// TwinCAT 3 PLC project mobject_graph
// Title: mobject-graph
// Company: mobject
// Author: mobject dev team
// ProjectVersion: 0.12.0
// ProgramVersion: 3.1.4024.0
// libraries:
//   Tc2_Standard, * (Beckhoff Automation GmbH)
//   Tc2_System, * (Beckhoff Automation GmbH)
//   Tc2_Utilities, * (Beckhoff Automation GmbH)
//   mobject-core,0.4.0,mobject
//   mobject-server,0.14.0,mobject
// project tree:
//   Alarms/Base/ Alarm.TcPOU
//   Alarms/ DeserializationFailedAlarm.TcPOU, DeserializationFailedNodeNotSupportedAlarm.TcPOU, FunctionFailedAlarm.TcPOU
//   Alarms/Events/ AlarmAddedEvent.TcPOU (not stored), I_AlarmAddedEvent.TcIO
//   Alarms/Host/ AlarmHost.TcPOU
//   Alarms/Interfaces/ I_Alarm.TcIO (not stored), I_Alarms.TcIO, I_HostAlarms.TcIO
//   API/ GraphFrameworkApi.TcPOU
//   API/Handlers/ CreateGraphMultiUserRpcHandler.TcPOU, CreateGraphRpcHandler.TcPOU, GetBlueprintsRpcHandler.TcPOU, GetContentValueHandler.TcPOU, UpdateParameterValueHandler.TcPOU, GetStatusRpcHandler.TcPOU
//   API/Visitors/ GetBlueprintsVisitor.TcPOU, GetStatusVisitor.TcPOU, IncludeInGetStatusVisitor.TcPOU, RetrieveNodeContentValue.TcPOU
//   Content/Base/ Content.TcPOU
//   Content/Events/ ContentAddedEvent.TcPOU (not stored), I_ContentAddedEvent.TcIO
//   Content/Host/ ContentHost.TcPOU
//   Content/Interface/ I_Content.TcIO (not stored), I_Contents.TcIO, I_HostContent.TcIO (not stored)
//   Errors/ MissingNodePrototypeDeserializationError.TcPOU (not stored)
//   Extensions/Base/ Extension.TcPOU
//   Extensions/Events/ ExtensionAddedEvent.TcPOU, I_ExtensionAddedEvent.TcIO (not stored)
//   Extensions/Host/ ExtensionHost.TcPOU
//   Extensions/Interface/ I_Extension.TcIO, I_Extensions.TcIO, I_HostExtensions.TcIO (not stored)
//   Extensions/Namespace/ ExtensionNamespace.TcPOU (not stored)
//   Extensions/PreExecutionCheck/Alarms/ PreExecutionCheckFailedAlarm.TcPOU
//   Extensions/PreExecutionCheck/Checks/ I_PreExecutionChecks.TcIO, PreExecutionChecks.TcPOU
//   Extensions/PreExecutionCheck/Interfaces/ I_PreCheckedNode.TcIO (not stored)
//   Extensions/PreExecutionCheck/ PreExecutionCheckExtension.TcPOU
//   GraphFramework/ GraphFramework.TcPOU
//   GraphFramework/Interface/ I_GraphFramework.TcIO
//   Graph/Base/ Graph.TcPOU
//   Graph/Events/ GraphAddedEvent.TcPOU (not stored), I_GraphAddedEvent.TcIO
//   Graph/Host/ GraphHost.TcPOU
//   Graph/Interfaces/ I_Graph.TcIO (not stored), I_Graphs.TcIO (not stored), I_HostGraphs.TcIO (not stored)
//   IecDatatypesPack/ IecDatatypesPack.TcPOU
//   InputPort/Base/ InputPort.TcPOU
//   InputPort/Events/ InputPortAddedEvent.TcPOU (not stored), InputPortChangedEvent.TcPOU (not stored), I_InputPortAddedEvent.TcIO (not stored), I_InputPortChangedEvent.TcIO (not stored)
//   InputPort/Host/ InputPortHost.TcPOU
//   InputPort/Interface/ I_HostInputPorts.TcIO, I_InputPort.TcIO (not stored), I_InputPorts.TcIO
//   Metadata/Base/ Metadata.TcPOU
//   Metadata/Events/ I_MetadataAddedEvent.TcIO, MetadataAddedEvent.TcPOU (not stored)
//   Metadata/Host/ MetadataHost.TcPOU
//   Metadata/Interface/ I_HostMetadata.TcIO, I_Metadata.TcIO, I_Metadatum.TcIO
//   NodeFactory/Base/ NodeFactory.TcPOU
//   NodeFactory/Datatype/ DatatypeNodeFactory.TcPOU
//   NodeFactory/Interface/ I_NodeFactory.TcIO (not stored)
//   NodePrototype/Base/ NodePrototype.TcPOU (not stored)
//   NodePrototype/Host/ NodePrototypeHost.TcPOU
//   NodePrototype/Interface/ I_NodePrototype.TcIO (not stored), I_NodePrototypes.TcIO
//   Node/Base/ Node.TcPOU
//   Node/Bundle/ AnyAliasArrayBundleNode.TcPOU, AnyStructureBundleNode.TcPOU, AnyArrayBundleNode.TcPOU, AnyAliasStructureBundleNode.TcPOU
//   Node/Events/ I_NodeAddedEvent.TcIO, I_NodeExecuteBeginEvent.TcIO, I_NodeExecuteEndEvent.TcIO, I_NodePreExecuteEvent.TcIO, NodeAddedEvent.TcPOU, NodeExecuteBeginEvent.TcPOU, NodeExecuteEndEvent.TcPOU, NodePreExecuteEvent.TcPOU
//   Node/Unbundle/ AnyAliasArrayUnbundleNode.TcPOU, AnyStructureUnbundleNode.TcPOU (not stored), AnyArrayUnbundleNode.TcPOU, AnyAliasStructureUnbundleNode.TcPOU
//   Node/Display/ AnyDisplayNode.TcPOU (not stored)
//   Node/Host/ NodeHost.TcPOU
//   Node/Interface/ I_HostNodes.TcIO (not stored), I_Node.TcIO, I_Nodes.TcIO
//   Node/Literal/ AnyLiteralNode.TcPOU (not stored)
//   OutputPort/Base/ OutputPort.TcPOU
//   OutputPort/Events/ I_OutputPortAddedEvent.TcIO, I_OutputPortChangedEvent.TcIO (not stored), OutputPortAddedEvent.TcPOU (not stored), OutputPortChangedEvent.TcPOU (not stored)
//   OutputPort/Host/ OutputPortHost.TcPOU
//   OutputPort/Interface/ I_HostOutputPorts.TcIO, I_OutputPort.TcIO (not stored), I_OutputPorts.TcIO
//   Packs/DatatypePack/ I_DatatypePack.TcIO (not stored)
//   Packs/GraphPack/ I_GraphPack.TcIO (not stored)
//   Packs/NodePack/ I_NodePack.TcIO
//   Parameters/Base/ Parameter.TcPOU
//   Parameters/Events/ I_ParameterAddedEvent.TcIO, ParameterAddedEvent.TcPOU
//   Parameters/Host/ ParameterHost.TcPOU
//   Parameters/Interface/ I_HostParameters.TcIO, I_Parameter.TcIO (not stored), I_Parameters.TcIO
//   Visitors/Interfaces/ I_AlarmVisitor.TcIO, I_ContentVisitor.TcIO, I_ExtensionVisitor.TcIO, I_GraphVisitor.TcIO, I_InputPortVisitor.TcIO (not stored), I_MetadataVisitor.TcIO (not stored), I_NodeFactoryVisitor.TcIO, I_NodePrototypeVisitor.TcIO (not stored), I_NodeVisitor.TcIO (not stored), I_OutputPortVisitor.TcIO (not stored), I_ParameterVisitor.TcIO

// ---- Alarms/Events/I_AlarmAddedEvent.TcIO
INTERFACE I_AlarmAddedEvent EXTENDS I_Event

PROPERTY PUBLIC Target : I_Alarm
GET
END_GET
END_PROPERTY

END_INTERFACE

// ---- Alarms/Interfaces/I_Alarms.TcIO
INTERFACE I_Alarms

METHOD PUBLIC Accept
VAR_INPUT
	Visitor : I_AlarmVisitor;
END_VAR
END_METHOD

METHOD AddAlarm
VAR_INPUT
	Alarm : I_Alarm;
END_VAR
END_METHOD

PROPERTY PUBLIC HasAlarms : BOOL
GET
END_GET
END_PROPERTY

PROPERTY PUBLIC HasRaisedAlarm : BOOL
GET
END_GET
END_PROPERTY

END_INTERFACE

// ---- Alarms/Interfaces/I_HostAlarms.TcIO
INTERFACE I_HostAlarms EXTENDS __SYSTEM.IQueryInterface

PROPERTY Alarms : I_Alarms
GET
END_GET
END_PROPERTY

END_INTERFACE

// ---- Content/Events/I_ContentAddedEvent.TcIO
INTERFACE I_ContentAddedEvent EXTENDS I_Event

PROPERTY PUBLIC Target : I_Content
GET
END_GET
END_PROPERTY

END_INTERFACE

// ---- Content/Interface/I_Contents.TcIO
INTERFACE I_Contents

METHOD PUBLIC Accept
VAR_INPUT
	visitor : I_ContentVisitor;
END_VAR
END_METHOD

METHOD AddContent
VAR_INPUT
	Content : I_Content;
END_VAR
END_METHOD

METHOD PUBLIC AddDataAsContent : I_Content
VAR_INPUT
	Name : T_MAXSTRING;
	Data : I_Datatype;
END_VAR
END_METHOD

PROPERTY PUBLIC HasContents : BOOL
GET
END_GET
END_PROPERTY

METHOD PUBLIC TryGetContentByName : BOOL
VAR_INPUT
	Name : T_MAXSTRING;
	Destination : REFERENCE TO I_Content;
END_VAR
END_METHOD

END_INTERFACE

// ---- Extensions/Interface/I_Extension.TcIO
INTERFACE I_Extension EXTENDS I_Disposable, I_HostContent, I_HostInputPorts, I_HostOutputPorts, I_HostAlarms, I_HostParameters, I_HostMetadata, I_EventEmitter, I_Deserializable, I_Serializable

METHOD PUBLIC Accept
VAR_INPUT
	Visitor : I_ExtensionVisitor;
END_VAR
END_METHOD

PROPERTY PUBLIC Name : T_MAXSTRING
GET
END_GET
END_PROPERTY

END_INTERFACE

// ---- Extensions/Interface/I_Extensions.TcIO
INTERFACE I_Extensions

METHOD PUBLIC Accept
VAR_INPUT
	Visitor : I_ExtensionVisitor;
END_VAR
END_METHOD

METHOD AddExtension
VAR_INPUT
	Extension : I_Extension;
END_VAR
END_METHOD

PROPERTY PUBLIC HasExtensions : BOOL
GET
END_GET
END_PROPERTY

METHOD PUBLIC TryGetExtensionByName : BOOL
VAR_INPUT
	Name : T_MAXSTRING;
	Destination : REFERENCE TO I_Extension;
END_VAR
END_METHOD

END_INTERFACE

// ---- Extensions/PreExecutionCheck/Checks/I_PreExecutionChecks.TcIO
INTERFACE I_PreExecutionChecks

METHOD PUBLIC Fail
VAR_INPUT
	Message : T_MAXSTRING;
END_VAR
END_METHOD

PROPERTY PUBLIC Failed : BOOL
GET
END_GET
END_PROPERTY

METHOD PUBLIC IsFalse
VAR_INPUT
	Actual : BOOL;
	Message : T_MAXSTRING;
END_VAR
END_METHOD

METHOD PUBLIC IsTrue
VAR_INPUT
	Actual : BOOL;
	Message : T_MAXSTRING;
END_VAR
END_METHOD

END_INTERFACE

// ---- GraphFramework/Interface/I_GraphFramework.TcIO
INTERFACE I_GraphFramework

METHOD PUBLIC Create : I_Graph
VAR_INPUT
END_VAR
END_METHOD

PROPERTY PUBLIC Datatypes : I_Datatypes
GET
END_GET
END_PROPERTY

PROPERTY PUBLIC NodeFactory : I_NodeFactory
GET
END_GET
END_PROPERTY

END_INTERFACE

// ---- Graph/Events/I_GraphAddedEvent.TcIO
INTERFACE I_GraphAddedEvent EXTENDS I_Event

PROPERTY PUBLIC Target : I_Graph
GET
END_GET
END_PROPERTY

END_INTERFACE

// ---- InputPort/Interface/I_HostInputPorts.TcIO
INTERFACE I_HostInputPorts EXTENDS __SYSTEM.IQueryInterface

PROPERTY InputPorts : I_InputPorts
GET
END_GET
END_PROPERTY

END_INTERFACE

// ---- InputPort/Interface/I_InputPorts.TcIO
INTERFACE I_InputPorts

METHOD PUBLIC Accept
VAR_INPUT
	Visitor : I_InputPortVisitor;
END_VAR
END_METHOD

METHOD PUBLIC AddDataAsInputPort : I_InputPort
VAR_INPUT
	Name : T_MAXSTRING;
	Data : I_Datatype;
END_VAR
END_METHOD

METHOD AddInputPort
VAR_INPUT
	InputPort : I_InputPort;
END_VAR
END_METHOD

PROPERTY PUBLIC HasInputPorts : BOOL
GET
END_GET
END_PROPERTY

METHOD PUBLIC TryGetInputPortByName : BOOL
VAR_INPUT
	Name : T_MAXSTRING;
	Destination : REFERENCE TO I_InputPort;
END_VAR
END_METHOD

END_INTERFACE

// ---- Metadata/Events/I_MetadataAddedEvent.TcIO
INTERFACE I_MetadataAddedEvent EXTENDS I_Event

PROPERTY PUBLIC Target : I_Metadata
GET
END_GET
END_PROPERTY

END_INTERFACE

// ---- Metadata/Interface/I_HostMetadata.TcIO
INTERFACE I_HostMetadata EXTENDS __SYSTEM.IQueryInterface

METHOD PUBLIC AddMetadata : I_HostMetadata
VAR_INPUT
	Name : T_MAXSTRING;
	Data : I_Datatype;
END_VAR
END_METHOD

PROPERTY Metadatum : I_Metadatum
GET
END_GET
END_PROPERTY

END_INTERFACE

// ---- Metadata/Interface/I_Metadata.TcIO
INTERFACE I_Metadata EXTENDS I_Disposable, I_Serializable

METHOD PUBLIC Accept
VAR_INPUT
	Visitor : I_MetadataVisitor;
END_VAR
END_METHOD

PROPERTY PUBLIC Data : I_DataType
GET
END_GET
END_PROPERTY

PROPERTY PUBLIC Name : T_MAXSTRING
GET
END_GET
END_PROPERTY

METHOD PUBLIC SerializeWith
VAR_INPUT
	Serializer : I_Serializer;
END_VAR
END_METHOD

END_INTERFACE

// ---- Metadata/Interface/I_Metadatum.TcIO
INTERFACE I_Metadatum

METHOD PUBLIC Accept
VAR_INPUT
	Visitor : I_MetadataVisitor;
END_VAR
END_METHOD

METHOD PUBLIC AddDataAsMetadata : I_Metadata
VAR_INPUT
	Name : T_MAXSTRING;
	Data : I_Datatype;
END_VAR
END_METHOD

METHOD AddMetadata
VAR_INPUT
	Metadata : I_Metadata;
END_VAR
END_METHOD

PROPERTY PUBLIC HasMetadata : BOOL
GET
END_GET
END_PROPERTY

METHOD PUBLIC TryGetMetadataByName : BOOL
VAR_INPUT
	Name : T_MAXSTRING;
	Destination : REFERENCE TO I_Metadata;
END_VAR
END_METHOD

END_INTERFACE

// ---- NodePrototype/Interface/I_NodePrototypes.TcIO
INTERFACE I_NodePrototypes

METHOD PUBLIC Accept
VAR_INPUT
	Visitor : I_NodePrototypeVisitor;
END_VAR
END_METHOD

PROPERTY PUBLIC HasNodePrototypes : BOOL
GET
END_GET
END_PROPERTY

END_INTERFACE

// ---- Node/Events/I_NodeAddedEvent.TcIO
INTERFACE I_NodeAddedEvent EXTENDS I_Event

PROPERTY PUBLIC Target : I_Node
GET
END_GET
END_PROPERTY

END_INTERFACE

// ---- Node/Events/I_NodeExecuteBeginEvent.TcIO
INTERFACE I_NodeExecuteBeginEvent EXTENDS I_Event

PROPERTY PUBLIC CpuCounterHighBytes : UDINT
GET
END_GET
END_PROPERTY

PROPERTY PUBLIC CpuCounterLowBytes : UDINT
GET
END_GET
END_PROPERTY

PROPERTY PUBLIC Target : I_Node
GET
END_GET
END_PROPERTY

END_INTERFACE

// ---- Node/Events/I_NodeExecuteEndEvent.TcIO
INTERFACE I_NodeExecuteEndEvent EXTENDS I_Event

PROPERTY PUBLIC Target : I_Node
GET
END_GET
END_PROPERTY

END_INTERFACE

// ---- Node/Events/I_NodePreExecuteEvent.TcIO
INTERFACE I_NodePreExecuteEvent EXTENDS I_Event

METHOD PUBLIC Cancel
VAR_INPUT
END_VAR
END_METHOD

PROPERTY PUBLIC ExecuteCancelled : BOOL
GET
END_GET
END_PROPERTY

PROPERTY PUBLIC Target : I_Node
GET
END_GET
END_PROPERTY

END_INTERFACE

// ---- Node/Interface/I_Node.TcIO
INTERFACE I_Node EXTENDS I_Disposable, I_HostContent, I_HostInputPorts, I_HostOutputPorts, I_HostAlarms, I_HostParameters, I_HostExtensions, I_HostMetadata, I_EventEmitter, I_Deserializable, I_Serializable

METHOD PUBLIC Accept
VAR_INPUT
	Visitor : I_NodeVisitor;
END_VAR
END_METHOD

METHOD Clone : I_Node
VAR_INPUT
END_VAR
END_METHOD

METHOD PUBLIC Execute
END_METHOD

PROPERTY PUBLIC Id : T_MAXSTRING
GET
END_GET
END_PROPERTY

PROPERTY PUBLIC Mode : DINT
GET
END_GET
END_PROPERTY

PROPERTY PUBLIC Order : DINT
GET
END_GET
END_PROPERTY

END_INTERFACE

// ---- Node/Interface/I_Nodes.TcIO
INTERFACE I_Nodes

METHOD PUBLIC Accept
VAR_INPUT
	Visitor : I_NodeVisitor;
END_VAR
END_METHOD

METHOD AddNode
VAR_INPUT
	Node : I_Node;
END_VAR
END_METHOD

PROPERTY PUBLIC HasNodes : BOOL
GET
END_GET
END_PROPERTY

METHOD PUBLIC TryGetNodeById : BOOL
VAR_INPUT
	Id : T_MAXSTRING;
	Destination : REFERENCE TO I_Node;
END_VAR
END_METHOD

END_INTERFACE

// ---- OutputPort/Events/I_OutputPortAddedEvent.TcIO
INTERFACE I_OutputPortAddedEvent extends I_Event

PROPERTY PUBLIC Target : I_OutputPort
GET
END_GET
END_PROPERTY

END_INTERFACE

// ---- OutputPort/Interface/I_HostOutputPorts.TcIO
INTERFACE I_HostOutputPorts EXTENDS __SYSTEM.IQueryInterface

PROPERTY OutputPorts : I_OutputPorts
GET
END_GET
END_PROPERTY

END_INTERFACE

// ---- OutputPort/Interface/I_OutputPorts.TcIO
INTERFACE I_OutputPorts

METHOD PUBLIC Accept
VAR_INPUT
	Visitor : I_OutputPortVisitor;
END_VAR
END_METHOD

METHOD PUBLIC AddDataAsOutputPort : I_OutputPort
VAR_INPUT
	Name : T_MAXSTRING;
	Data : I_Datatype;
END_VAR
END_METHOD

METHOD AddOutputPort
VAR_INPUT
	OutputPort : I_OutputPort;
END_VAR
END_METHOD

PROPERTY PUBLIC HasOutputPorts : BOOL
GET
END_GET
END_PROPERTY

METHOD PUBLIC TryGetOutputPortByName : BOOL
VAR_INPUT
	Name : T_MAXSTRING;
	Destination : REFERENCE TO I_OutputPort;
END_VAR
END_METHOD

END_INTERFACE

// ---- Packs/NodePack/I_NodePack.TcIO
INTERFACE I_NodePack

METHOD PUBLIC RegisterWithNodeFactory
VAR_INPUT
	NodeFactory : I_NodeFactory;
END_VAR
END_METHOD

END_INTERFACE

// ---- Parameters/Events/I_ParameterAddedEvent.TcIO
INTERFACE I_ParameterAddedEvent EXTENDS I_Event

PROPERTY PUBLIC TargetParameter : I_Parameter
GET
END_GET
END_PROPERTY

END_INTERFACE

// ---- Parameters/Interface/I_HostParameters.TcIO
INTERFACE I_HostParameters EXTENDS __SYSTEM.IQueryInterface

PROPERTY Parameters : I_Parameters
GET
END_GET
END_PROPERTY

END_INTERFACE

// ---- Parameters/Interface/I_Parameters.TcIO
INTERFACE I_Parameters

METHOD PUBLIC Accept
VAR_INPUT
	Visitor : I_ParameterVisitor;
END_VAR
END_METHOD

METHOD PUBLIC AddDataAsParameter : I_Parameter
VAR_INPUT
	Name : T_MAXSTRING;
	Data : I_Datatype;
END_VAR
END_METHOD

METHOD AddParameter
VAR_INPUT
	Parameter : I_Parameter;
END_VAR
END_METHOD

METHOD PUBLIC TryGetParameterByName : BOOL
VAR_INPUT
	Name : T_MAXSTRING;
	Destination : REFERENCE TO I_Parameter;
END_VAR
END_METHOD

END_INTERFACE

// ---- Visitors/Interfaces/I_AlarmVisitor.TcIO
INTERFACE I_AlarmVisitor

METHOD VisitError
VAR_INPUT
	VisitingError : I_Alarm;
END_VAR
END_METHOD

END_INTERFACE

// ---- Visitors/Interfaces/I_ContentVisitor.TcIO
INTERFACE I_ContentVisitor

METHOD VisitContent
VAR_INPUT
	VisitingContent : I_Content;
END_VAR
END_METHOD

END_INTERFACE

// ---- Visitors/Interfaces/I_ExtensionVisitor.TcIO
INTERFACE I_ExtensionVisitor

METHOD VisitExtension
VAR_INPUT
	VisitingExtension : I_Extension;
END_VAR
END_METHOD

END_INTERFACE

// ---- Visitors/Interfaces/I_GraphVisitor.TcIO
INTERFACE I_GraphVisitor

METHOD VisitGraph
VAR_INPUT
	VisitingGraph : I_Graph;
END_VAR
END_METHOD

END_INTERFACE

// ---- Visitors/Interfaces/I_NodeFactoryVisitor.TcIO
INTERFACE I_NodeFactoryVisitor

METHOD VisitNodeFactory
VAR_INPUT
	VisitingNodeFactory : I_NodeFactory;
END_VAR
END_METHOD

END_INTERFACE

// ---- Visitors/Interfaces/I_ParameterVisitor.TcIO
INTERFACE I_ParameterVisitor

METHOD VisitParameter
VAR_INPUT
	VisitingProperty : I_Parameter;
END_VAR
END_METHOD

END_INTERFACE

// ---- Alarms/Base/Alarm.TcPOU
{attribute 'linkalways'} 
{attribute 'no_explicit_call' := 'This FB is a CLASS and must be accessed using methods or properties'}
{attribute 'enable_dynamic_creation'}
FUNCTION_BLOCK ABSTRACT Alarm IMPLEMENTS I_Alarm

METHOD PUBLIC Accept
VAR_INPUT
	Visitor : I_AlarmVisitor;
END_VAR
Visitor.VisitAlarm(this^);
END_METHOD

PROPERTY ABSTRACT Active : BOOL
GET
END_GET
END_PROPERTY

METHOD ABSTRACT Clear
END_METHOD

METHOD FB_init : BOOL
VAR_INPUT
	bInitRetains : BOOL; // if TRUE, the retain variables are initialized (warm start / cold start)
	bInCopyCode : BOOL;  // if TRUE, the instance afterwards gets moved into the copy code (online change)
	Parent : I_HostAlarms;
END_VAR
RegisterWithParent(Parent);
END_METHOD

PROPERTY ABSTRACT Message : T_MaxString
GET
END_GET
END_PROPERTY

PROPERTY ABSTRACT Reason : T_MaxString
GET
END_GET
END_PROPERTY

METHOD RegisterWithParent
VAR_INPUT
	Parent : I_HostAlarms;
END_VAR
IF Parent = 0 THEN
	RETURN;
END_IF

Parent.Alarms.AddAlarm(THIS^);
END_METHOD

METHOD PUBLIC SerializeWith
VAR_INPUT
	Serializer : I_Serializer;
END_VAR
VAR
	isActive : BOOL := Active;
	errorMessage : T_MAXSTRING := Message;
	reasonMessage : T_MAXSTRING := Reason;
END_VAR
Serializer.StartObject();
Serializer.AddKeyString('message',errorMessage);
Serializer.AddKeyBool('active',isActive);

IF reasonMessage <> '' THEN
	Serializer.AddKeyString('reason',reasonMessage);
END_IF

Serializer.EndObject();
END_METHOD

END_FUNCTION_BLOCK

// ---- Alarms/DeserializationFailedAlarm.TcPOU
{attribute 'linkalways'} 
{attribute 'no_explicit_call' := 'This FB is a CLASS and must be accessed using methods or properties'}
{attribute 'enable_dynamic_creation'}
FUNCTION_BLOCK PUBLIC DeserializationFailedAlarm EXTENDS Alarm
VAR
	state : (CLEARED, RAISED);
	_reason : T_MAXSTRING;
END_VAR

PROPERTY Active : BOOL
GET
Active := state <> CLEARED;
END_GET
END_PROPERTY

METHOD PUBLIC Clear
_reason := '';
state := CLEARED;
END_METHOD

PROPERTY PUBLIC Message : T_MaxString
GET
Message := 'Deserialization failed';
END_GET
END_PROPERTY

METHOD PUBLIC Raise
VAR_INPUT
	Reason : T_MAXSTRING;
END_VAR
_reason := Reason;
state := RAISED;
END_METHOD

PROPERTY Reason : T_MaxString
GET
Reason := _reason;
END_GET
END_PROPERTY

END_FUNCTION_BLOCK

// ---- Alarms/DeserializationFailedNodeNotSupportedAlarm.TcPOU
{attribute 'linkalways'} 
{attribute 'no_explicit_call' := 'This FB is a CLASS and must be accessed using methods or properties'}
{attribute 'enable_dynamic_creation'}
FUNCTION_BLOCK PUBLIC DeserializationFailedNodeNotSupportedAlarm EXTENDS Alarm
VAR
	state : (CLEARED, RAISED);
	_reason : T_MAXSTRING;
END_VAR

PROPERTY Active : BOOL
GET
Active := state <> CLEARED;
END_GET
END_PROPERTY

METHOD PUBLIC Clear
_reason := '';
state := CLEARED;
END_METHOD

PROPERTY PUBLIC Message : T_MaxString
GET
Message := 'Node type is not installed';
END_GET
END_PROPERTY

METHOD PUBLIC Raise
VAR_INPUT
	NodeType : T_MAXSTRING;
END_VAR
_reason := NodeType;
state := RAISED;
END_METHOD

PROPERTY Reason : T_MaxString
GET
Reason := _reason;
END_GET
END_PROPERTY

END_FUNCTION_BLOCK

// ---- Node/Base/Node.TcPOU
{attribute 'linkalways'} 
{attribute 'no_explicit_call' := 'This FB is a CLASS and must be accessed using methods or properties'}
{attribute 'enable_dynamic_creation'}
FUNCTION_BLOCK ABSTRACT Node EXTENDS Disposable IMPLEMENTS I_Node
VAR
	_id : T_MAXSTRING;
	_order : DINT;
	_mode : DINT;
	eventEmitter : EventEmitter;
	inputPortHost : InputPortHost(THIS^, eventEmitter);
	outputPortHost : OutputPortHost(THIS^, eventEmitter);
	parameterHost : ParameterHost(THIS^, eventEmitter);
	contentHost : ContentHost(THIS^, eventEmitter);
	alarmHost : AlarmHost(THIS^, eventEmitter);
	metadataHost : MetadataHost(THIS^, eventEmitter);
	extensionHost : ExtensionHost(THIS^,eventEmitter);
	deserializationFailedAlarm : DeserializationFailedAlarm(THIS^);
END_VAR

METHOD PUBLIC Accept
VAR_INPUT
	Visitor : I_NodeVisitor;
END_VAR
Visitor.VisitNode(THIS^);
END_METHOD

METHOD PROTECTED AddContent : I_Content
VAR_INPUT
	Name : T_MAXSTRING;
	Data : I_Datatype;
END_VAR
AddContent := Contents.AddDataAsContent(Name, Data);
END_METHOD

METHOD PROTECTED AddInput : I_InputPort
VAR_INPUT
	Name : T_MAXSTRING;
	Data : I_Datatype;
END_VAR
AddInput := InputPorts.AddDataAsInputPort(Name, Data);
END_METHOD

METHOD PUBLIC AddMetadata : I_HostMetadata
VAR_INPUT
	Name : T_MAXSTRING;
	Data : I_Datatype;
END_VAR
Metadatum.AddDataAsMetadata(Name, Data);
AddMetadata := THIS^;
END_METHOD

METHOD PROTECTED AddOutput : I_OutputPort
VAR_INPUT
	Name : T_MAXSTRING;
	Data : I_Datatype;
END_VAR
AddOutput := OutputPorts.AddDataAsOutputPort(Name, Data);
END_METHOD

METHOD PROTECTED AddParameter : I_Parameter
VAR_INPUT
	Name : T_MAXSTRING;
	Data : I_Datatype;
END_VAR
AddParameter := Parameters.AddDataAsParameter(Name, Data);
END_METHOD

PROPERTY PUBLIC Alarms : I_Alarms
GET
Alarms := alarmHost;
END_GET
END_PROPERTY

METHOD PUBLIC ABSTRACT Clone : I_Node
VAR_INPUT
END_VAR
END_METHOD

PROPERTY PUBLIC Contents : I_Contents
GET
Contents := contentHost;
END_GET
END_PROPERTY

METHOD PRIVATE EmitNodeExecuteBeginEvent : BOOL;
VAR
	pNodeExecuteBeginEvent : POINTER TO NodeExecuteBeginEvent;
END_VAR
pNodeExecuteBeginEvent := __NEW(NodeExecuteBeginEvent(Target := THIS^));
eventEmitter.Emit('OnNodeExecuteBegin',pNodeExecuteBeginEvent^);
pNodeExecuteBeginEvent^.Dispose();
END_METHOD

METHOD PRIVATE EmitNodeExecuteEndEvent : BOOL;
VAR
	pNodeExecuteEndEvent : POINTER TO NodeExecuteEndEvent;
END_VAR
pNodeExecuteEndEvent := __NEW(NodeExecuteEndEvent(Target := THIS^));
eventEmitter.Emit('OnNodeExecuteEnd',pNodeExecuteEndEvent^);
pNodeExecuteEndEvent^.Dispose();
END_METHOD

METHOD PRIVATE EmitOnNodePreExecuteEvent : BOOL;
VAR_INPUT
	CancelRequested : REFERENCE TO BOOL;
END_VAR
VAR
	pNodePreExecuteEvent : POINTER TO NodePreExecuteEvent;
END_VAR
pNodePreExecuteEvent := __NEW(NodePreExecuteEvent(Target := THIS^));
eventEmitter.Emit('OnNodePreExecute',pNodePreExecuteEvent^);

IF pNodePreExecuteEvent^.ExecuteCancelled THEN
	CancelRequested := TRUE;
END_IF

pNodePreExecuteEvent^.Dispose();
END_METHOD

METHOD PUBLIC Execute
VAR
	cancelExecuteResponse : BOOL := FALSE;
END_VAR
EmitOnNodePreExecuteEvent(cancelExecuteResponse);

IF cancelExecuteResponse THEN
	RETURN;
END_IF

EmitNodeExecuteBeginEvent();
OnExecute();
EmitNodeExecuteEndEvent();
END_METHOD

PROPERTY PUBLIC Extensions : I_Extensions
GET
Extensions := extensionHost;
END_GET
END_PROPERTY

PROPERTY PUBLIC HasRaisedAlarm : BOOL
GET
HasRaisedAlarm := alarmHost.HasRaisedAlarm;
END_GET
END_PROPERTY

PROPERTY PUBLIC Id : T_MAXSTRING
GET
Id := _id;
END_GET
END_PROPERTY

PROPERTY PUBLIC InputPorts : I_InputPorts
GET
InputPorts := inputPortHost;
END_GET
END_PROPERTY

PROPERTY PUBLIC Metadatum : I_Metadatum
GET
Metadatum := metadataHost;
END_GET
END_PROPERTY

PROPERTY PUBLIC Mode : DINT
GET
Mode := _mode;
END_GET
END_PROPERTY

METHOD PUBLIC OffEvent
VAR_INPUT
	EventName : T_MaxString;
	EventHandler : I_EventHandler;
END_VAR
eventEmitter.OffEvent(EventName, EventHandler);
END_METHOD

METHOD PUBLIC OnceEvent
VAR_INPUT
	EventName : T_MaxString;
	EventHandler : I_EventHandler;
END_VAR
eventEmitter.OnceEvent(EventName, EventHandler);
END_METHOD

METHOD PUBLIC OnEvent
VAR_INPUT
	EventName : T_MaxString;
	EventHandler : I_EventHandler;
END_VAR
eventEmitter.OnEvent(EventName, EventHandler);
END_METHOD

METHOD PROTECTED ABSTRACT OnExecute : HRESULT
END_METHOD

PROPERTY PUBLIC Order : DINT
GET
Order := _order;
END_GET
END_PROPERTY

PROPERTY PUBLIC OutputPorts : I_OutputPorts
GET
OutputPorts := outputPortHost;
END_GET
END_PROPERTY

PROPERTY PUBLIC Parameters : I_Parameters
GET
Parameters := parameterHost;
END_GET
END_PROPERTY

PROPERTY PUBLIC Self : I_Node
GET
Self := This^;
END_GET
END_PROPERTY

METHOD PUBLIC SerializeWith
VAR_INPUT
	Serializer : I_Serializer;
END_VAR
Serializer.StartObject();
Serializer.AddKeyString('id',_id);
Serializer.AddKeyDint('order',_order);
Serializer.AddKeyDint('mode',_mode);
inputPortHost.SerializeWith(Serializer);
outputPortHost.SerializeWith(Serializer);
parameterHost.SerializeWith(Serializer);
contentHost.SerializeWith(Serializer);
alarmHost.SerializeWith(Serializer);
extensionHost.SerializeWith(Serializer);
metadataHost.SerializeWith(Serializer);
Serializer.EndObject();
END_METHOD

METHOD PUBLIC TryDeserializeFrom : BOOL
VAR_INPUT
	Deserializer : I_Deserializer;
	Feedback : I_DeserializerFeedback;
END_VAR
DeserializationFailedAlarm.Clear();

IF NOT Deserializer.TryGetKeyString('id', _id, Feedback) THEN
	DeserializationFailedAlarm.Raise('Missing node id');	
	RETURN;
END_IF

IF NOT Deserializer.TryGetKeyDint('order', _order, Feedback) THEN
	DeserializationFailedAlarm.Raise('Missing node order');	
	RETURN;
END_IF

IF NOT Deserializer.TryGetKeyDint('mode', _mode, Feedback) THEN
	DeserializationFailedAlarm.Raise('Missing node mode');	
	RETURN;
END_IF

IF NOT parameterHost.TryDeserializeFrom(Deserializer, Feedback) THEN
	DeserializationFailedAlarm.Raise('Failed to deserialize parameters');	
	RETURN;
END_IF

IF NOT extensionHost.TryDeserializeFrom(Deserializer, Feedback) THEN
	DeserializationFailedAlarm.Raise('Failed to deserialize extensions');	
	RETURN;
END_IF

TryDeserializeFrom := TRUE;
END_METHOD

END_FUNCTION_BLOCK

// ---- InputPort/Host/InputPortHost.TcPOU
{attribute 'linkalways'} 
{attribute 'no_explicit_call' := 'This FB is a CLASS and must be accessed using methods or properties'}
{attribute 'enable_dynamic_creation'}
FUNCTION_BLOCK InputPortHost IMPLEMENTS I_InputPorts, I_Serializable
VAR
	hostParent : I_HostInputPorts;
	eventTarget : I_EventTarget;
	ports : OrderedDictionary;
	selfCreatedInputPorts : Stack;
END_VAR

METHOD PUBLIC Accept
VAR_INPUT
	Visitor : I_InputPortVisitor;
END_VAR
VAR
	enumerator : I_ForwardEnumerator;
	port : I_InputPort;
END_VAR
enumerator := ports.GetEnumerator();

WHILE (enumerator.MoveNext()) DO
	
	IF enumerator.TryGet(port) THEN
		port.Accept(Visitor);
	END_IF

END_WHILE

enumerator.Dispose();
END_METHOD

METHOD PUBLIC AddDataAsInputPort : I_InputPort
VAR_INPUT
	Name : T_MAXSTRING;
	Data : I_Datatype;
END_VAR
VAR
	port : I_InputPort;
END_VAR
port := CreateInputPort(Name, Data);
selfCreatedInputPorts.Push(port);
AddDataAsInputPort := port;
END_METHOD

METHOD PUBLIC AddInputPort
VAR_INPUT
	InputPort : I_InputPort;
END_VAR
ports.AddOrUpdate(InputPort.Name, InputPort);
EmitOnPortAddedEvent(InputPort);
END_METHOD

METHOD PRIVATE CreateInputPort : I_InputPort
VAR_INPUT
	PortName : T_MAXSTRING;
	PortData : I_Datatype;
END_VAR
VAR
	pPort : POINTER TO InputPort;
END_VAR
pPort := __NEW(InputPort(Name := PortName, Data := PortData, Parent := hostParent));
CreateInputPort := pPort^;
END_METHOD

METHOD PRIVATE DisposeSelfCreatedInputPorts : BOOL
VAR
	port : I_InputPort;
END_VAR
WHILE selfCreatedInputPorts.TryPop(port) DO
	port.Dispose();
END_WHILE
END_METHOD

METHOD PROTECTED EmitOnPortAddedEvent
VAR_INPUT
	Port : I_InputPort;
END_VAR
VAR
	pInputPortAddedEvent : POINTER TO InputPortAddedEvent;
END_VAR
IF eventTarget = 0 THEN
	RETURN;
END_IF

pInputPortAddedEvent := __NEW(InputPortAddedEvent(Target := Port));
eventTarget.Emit('OnInputPortAdded',pInputPortAddedEvent^);
pInputPortAddedEvent^.Dispose();
END_METHOD

METHOD FB_exit : BOOL
VAR_INPUT
	bInCopyCode : BOOL; // if TRUE, the exit method is called for exiting an instance that is copied afterwards (online change).
END_VAR
IF bInCopyCode THEN
	RETURN;
END_IF

DisposeSelfCreatedInputPorts();
END_METHOD

METHOD FB_init : BOOL
VAR_INPUT
	bInitRetains : BOOL; // if TRUE, the retain variables are initialized (warm start / cold start)
	bInCopyCode : BOOL;  // if TRUE, the instance afterwards gets moved into the copy code (online change)
	Parent : I_HostInputPorts;
	parentEventTarget : I_EventTarget;
END_VAR
hostParent := Parent;
eventTarget := parentEventTarget;
END_METHOD

PROPERTY PUBLIC HasInputPorts : BOOL
GET
HasInputPorts := NOT ports.IsEmpty;
END_GET
END_PROPERTY

METHOD PUBLIC SerializeWith
VAR_INPUT
	Serializer : I_Serializer;
END_VAR
VAR
	enumerator : I_ForwardEnumerator;
	port : I_InputPort;
END_VAR
IF ports.Count = 0 THEN
	RETURN;
END_IF

Serializer.AddKey('inputPorts');
Serializer.StartArray();

enumerator := ports.GetEnumerator();

WHILE enumerator.MoveNext() DO
	IF enumerator.TryGet(port) THEN
		port.SerializeWith(Serializer);
	END_IF
END_WHILE

Serializer.EndArray();
enumerator.Dispose();
END_METHOD

METHOD PUBLIC TryGetInputPortByName : BOOL
VAR_INPUT
	Name : T_MAXSTRING;
	Destination : REFERENCE TO I_InputPort;
END_VAR
VAR
	port : I_InputPort;
END_VAR
IF NOT ports.TryGetValue(Name, port) THEN
	RETURN;
END_IF

Destination := port;
TryGetInputPortByName := TRUE;
END_METHOD

END_FUNCTION_BLOCK

// ---- InputPort/Base/InputPort.TcPOU
{attribute 'linkalways'} 
{attribute 'no_explicit_call' := 'This FB is a CLASS and must be accessed using methods or properties'}
{attribute 'enable_dynamic_creation'}
FUNCTION_BLOCK InputPort EXTENDS Disposable IMPLEMENTS I_InputPort
VAR
	_name : T_MAXSTRING;
	_data : I_Datatype;
	_connectedTo : I_OutputPort;
	parent : I_HostInputPorts;
	eventEmitter : EventEmitter;
	metadataHost : MetadataHost(THIS^, eventEmitter);
END_VAR

METHOD PUBLIC Accept
VAR_INPUT
	Visitor : I_InputPortVisitor;
END_VAR
Visitor.VisitInputPort(THIS^);
END_METHOD

METHOD PUBLIC AddMetadata : I_HostMetadata
VAR_INPUT
	Name : T_MAXSTRING;
	Data : I_Datatype;
END_VAR
Metadatum.AddDataAsMetadata(Name, Data);
AddMetadata := THIS^;
END_METHOD

PROPERTY PUBLIC Connected : BOOL
GET
Connected := _connectedTo <> 0;
END_GET
END_PROPERTY

PROPERTY PUBLIC Data : I_Datatype
GET
Data := _data;
END_GET
END_PROPERTY

METHOD PUBLIC Disconnect
IF NOT Connected THEN
	RETURN;
END_IF

_connectedTo.OffEvent('OnOutputPortChanged', THIS^);
_connectedTo := 0;
_data.ClearReference();
END_METHOD

METHOD PROTECTED EmitOnInputPortChanged
VAR_INPUT
	PortChanged : I_InputPort;
END_VAR
VAR
	pInputPortChangeEvent : POINTER TO InputPortChangedEvent;
END_VAR
pInputPortChangeEvent := __NEW(InputPortChangedEvent(Target := PortChanged));
eventEmitter.Emit('OnInputPortChanged',pInputPortChangeEvent^);
pInputPortChangeEvent^.Dispose();
END_METHOD

METHOD FB_init : BOOL
VAR_INPUT
	bInitRetains : BOOL; // if TRUE, the retain variables are initialized (warm start / cold start)
	bInCopyCode : BOOL;  // if TRUE, the instance afterwards gets moved into the copy code (online change)
	Name : T_MAXSTRING;
	Data : I_Datatype;
	Parent : I_HostInputPorts;
END_VAR
_name := Name;
_data := Data;
RegisterWithParent(Parent);
END_METHOD

METHOD PUBLIC HandleEvent
VAR_INPUT
	Event : I_Event;
END_VAR
VAR
	outputPortChangedEvent : I_OutputPortChangedEvent;
END_VAR
IF __QUERYINTERFACE(Event, outputPortChangedEvent) THEN
	HandleOutputPortChangedEvent(outputPortChangedEvent.Target);
END_IF
END_METHOD

METHOD PROTECTED HandleOutputPortChangedEvent
VAR_INPUT
	Source : I_OutputPort;
END_VAR
EmitOnInputPortChanged(THIS^);
END_METHOD

PROPERTY PUBLIC Metadatum : I_Metadatum
GET
Metadatum := metadataHost;
END_GET
END_PROPERTY

PROPERTY PUBLIC Name : T_MAXSTRING
GET
Name := _name;
END_GET
END_PROPERTY

METHOD PUBLIC OffEvent
VAR_INPUT
	EventName : T_MaxString;
	EventHandler : I_EventHandler;
END_VAR
eventEmitter.OffEvent(EventName, EventHandler);
END_METHOD

METHOD PUBLIC OnceEvent
VAR_INPUT
	EventName : T_MaxString;
	EventHandler : I_EventHandler;
END_VAR
eventEmitter.OnceEvent(EventName, EventHandler);
END_METHOD

METHOD PUBLIC OnEvent
VAR_INPUT
	EventName : T_MaxString;
	EventHandler : I_EventHandler;
END_VAR
eventEmitter.OnEvent(EventName, EventHandler);
END_METHOD

METHOD PUBLIC RegisterWithParent
VAR_INPUT
	Parent : I_HostInputPorts;
END_VAR
IF Parent = 0 THEN
	RETURN;
END_IF

THIS^.parent := Parent;
Parent.InputPorts.AddInputPort(THIS^);
END_METHOD

METHOD PUBLIC SerializeWith
VAR_INPUT
	Serializer : I_Serializer;
END_VAR
VAR 
	isConnected : BOOL := Connected;
END_VAR
Serializer.StartObject();
Serializer.AddKeyString('name',_name);
Serializer.AddKeyBool('connected',isConnected);
Serializer.Addkey('datatype');
_data.SerializeTypeWith(Serializer);
Serializer.AddkeyObject('value',_data);
metadataHost.SerializeWith(Serializer);
Serializer.EndObject();
END_METHOD

METHOD PUBLIC TryConnectTo : BOOL
VAR_INPUT
	OutputPort : I_OutputPort;
END_VAR
IF NOT _data.TryMakeReferenceTo(OutputPort.Data) THEN
	RETURN;
END_IF

_connectedTo := OutputPort;
_connectedTo.OnEvent('OnOutputPortChanged', THIS^);
TryConnectTo := TRUE;
END_METHOD

END_FUNCTION_BLOCK

// ---- Metadata/Host/MetadataHost.TcPOU
{attribute 'linkalways'} 
{attribute 'no_explicit_call' := 'This FB is a CLASS and must be accessed using methods or properties'}
{attribute 'enable_dynamic_creation'}
FUNCTION_BLOCK MetadataHost IMPLEMENTS I_Metadatum, I_Serializable
VAR
	hostParent : I_HostMetadata;
	eventTarget : I_EventTarget;
	meta : OrderedDictionary;
	selfCreatedMetadata : Stack;
END_VAR

METHOD PUBLIC Accept
VAR_INPUT
	Visitor : I_MetadataVisitor;
END_VAR
VAR
	enumerator : I_ForwardEnumerator;
	metadata : I_Metadata;
END_VAR
enumerator := meta.GetEnumerator();

WHILE (enumerator.MoveNext()) DO
	
	IF enumerator.TryGet(metadata) THEN
		metadata.Accept(Visitor);
	END_IF

END_WHILE

enumerator.Dispose();
END_METHOD

METHOD PUBLIC AddDataAsMetadata : I_Metadata
VAR_INPUT
	Name : T_MAXSTRING;
	Data : I_Datatype;
END_VAR
VAR
	metadata : I_Metadata;
END_VAR
metadata := CreateMetadata(Name, Data);
selfCreatedMetadata.Push(metadata);
AddDataAsMetadata := metadata;
END_METHOD

METHOD PUBLIC AddMetadata
VAR_INPUT
	Metadata : I_Metadata;
END_VAR
meta.AddOrUpdate(Metadata.Name, Metadata);
EmitOnMetadataAddedEvent(Metadata);
END_METHOD

METHOD PRIVATE CreateMetadata : I_Metadata
VAR_INPUT
	MetadataName : T_MAXSTRING;
	MetadataData : I_Datatype;
END_VAR
VAR
	pMetadata : POINTER TO Metadata;
END_VAR
pMetadata := __NEW(Metadata(Name := MetadataName, Data := MetadataData, Parent := hostParent));
CreateMetadata := pMetadata^;
END_METHOD

METHOD PROTECTED DisposeSelfCreatedMetadata : BOOL
VAR
	metadata : I_Metadata;
END_VAR
WHILE selfCreatedMetadata.TryPop(metadata) DO
	metadata.Dispose();
END_WHILE
END_METHOD

METHOD PROTECTED EmitOnMetadataAddedEvent
VAR_INPUT
	Metadata : I_Metadata;
END_VAR
VAR
	pMetadataAddedEvent : POINTER TO MetadataAddedEvent;
END_VAR
IF eventTarget = 0 THEN
	RETURN;
END_IF

pMetadataAddedEvent := __NEW(MetadataAddedEvent(Target := Metadata));
eventTarget.Emit('OnMetadataAdded',pMetadataAddedEvent^);
pMetadataAddedEvent^.Dispose();
END_METHOD

METHOD FB_exit : BOOL
VAR_INPUT
	bInCopyCode : BOOL; // if TRUE, the exit method is called for exiting an instance that is copied afterwards (online change).
END_VAR
IF bInCopyCode THEN
	RETURN;
END_IF

DisposeSelfCreatedMetadata();
END_METHOD

METHOD FB_init : BOOL
VAR_INPUT
	bInitRetains : BOOL; // if TRUE, the retain variables are initialized (warm start / cold start)
	bInCopyCode : BOOL;  // if TRUE, the instance afterwards gets moved into the copy code (online change)
	Parent : I_HostMetadata;
	ParentEventTarget : I_EventTarget;
END_VAR
hostParent := Parent;
eventTarget := ParentEventTarget;
END_METHOD

PROPERTY PUBLIC HasMetadata : BOOL
GET
HasMetadata := NOT meta.IsEmpty;
END_GET
END_PROPERTY

METHOD PUBLIC SerializeWith
VAR_INPUT
	Serializer : I_Serializer;
END_VAR
VAR
	enumerator : I_ForwardEnumerator;
	metadata : I_Metadata;
END_VAR
IF meta.Count = 0 THEN
	RETURN;
END_IF

Serializer.AddKey('metadata');
Serializer.StartArray();

enumerator := meta.GetEnumerator();

WHILE enumerator.MoveNext() DO
	IF enumerator.TryGet(metadata) THEN
		metadata.SerializeWith(Serializer);
	END_IF
END_WHILE

Serializer.EndArray();
enumerator.Dispose();
END_METHOD

METHOD PUBLIC TryGetMetadataByName : BOOL
VAR_INPUT
	Name : T_MAXSTRING;
	Destination : REFERENCE TO I_Metadata;
END_VAR
VAR
	metadata : I_Metadata;
END_VAR
IF NOT meta.TryGetValue(Name, metadata) THEN
	RETURN;
END_IF

Destination := metadata;
TryGetMetadataByName := TRUE;
END_METHOD

END_FUNCTION_BLOCK

// ---- Metadata/Base/Metadata.TcPOU
{attribute 'linkalways'} 
{attribute 'no_explicit_call' := 'This FB is a CLASS and must be accessed using methods or properties'}
{attribute 'enable_dynamic_creation'}
FUNCTION_BLOCK Metadata EXTENDS Disposable IMPLEMENTS I_Metadata
VAR
	_name : T_MAXSTRING;
	_data : I_Datatype;
	_parent : I_HostMetadata;
END_VAR

METHOD PUBLIC Accept
VAR_INPUT
	Visitor : I_MetadataVisitor;
END_VAR
Visitor.VisitMetadatum(this^);
END_METHOD

PROPERTY PUBLIC Data : I_DataType
GET
Data := _data;
END_GET
END_PROPERTY

METHOD FB_init : BOOL
VAR_INPUT
	bInitRetains : BOOL; // if TRUE, the retain variables are initialized (warm start / cold start)
	bInCopyCode : BOOL;  // if TRUE, the instance afterwards gets moved into the copy code (online change)
	Name : T_MAXSTRING;
	Data : I_Datatype;
	Parent : I_HostMetadata;
END_VAR
_name := Name;
_data := Data;
RegisterWithParent(Parent);
END_METHOD

PROPERTY PUBLIC Name : T_MAXSTRING
GET
Name := _name;
END_GET
END_PROPERTY

PROPERTY PUBLIC Parent : I_HostMetadata
GET
Parent := _parent;
END_GET
END_PROPERTY

METHOD PUBLIC RegisterWithParent
VAR_INPUT
	Parent : I_HostMetadata;
END_VAR
IF Parent = 0 THEN
	RETURN;
END_IF

THIS^._parent := Parent;
Parent.Metadatum.AddMetadata(THIS^);
END_METHOD

METHOD PUBLIC SerializeWith
VAR_INPUT
	Serializer : I_Serializer;
END_VAR
Serializer.StartObject();
Serializer.AddKeyString('name',_name);
Serializer.Addkey('datatype');
_data.SerializeTypeWith(Serializer);
Serializer.AddkeyObject('value',_data);
Serializer.EndObject();
END_METHOD

END_FUNCTION_BLOCK

// ---- OutputPort/Base/OutputPort.TcPOU
{attribute 'linkalways'} 
{attribute 'no_explicit_call' := 'This FB is a CLASS and must be accessed using methods or properties'}
{attribute 'enable_dynamic_creation'}
FUNCTION_BLOCK OutputPort EXTENDS Disposable IMPLEMENTS I_OutputPort
VAR
	_name : T_MAXSTRING;
	_data : I_Datatype;
	parent : I_HostOutputPorts;
	eventEmitter : EventEmitter;
	metadataHost : MetadataHost(THIS^, eventEmitter);
END_VAR

METHOD PUBLIC Accept
VAR_INPUT
	Visitor : I_OutputPortVisitor;
END_VAR
Visitor.VisitOutputPort(THIS^);
END_METHOD

METHOD PUBLIC AddMetadata : I_HostMetadata
VAR_INPUT
	Name : T_MAXSTRING;
	Data : I_Datatype;
END_VAR
Metadatum.AddDataAsMetadata(Name, Data);
AddMetadata := THIS^;
END_METHOD

PROPERTY PUBLIC Data : I_Datatype
GET
Data := _data;
END_GET
END_PROPERTY

METHOD Protected EmitOnOutputPortChangeEvent
VAR_INPUT
	PortChanged : I_OutputPort;
END_VAR
VAR
	pOutputPortChangeEvent : POINTER TO OutputPortChangedEvent;
END_VAR
pOutputPortChangeEvent := __NEW(OutputPortChangedEvent(Target := PortChanged));
eventEmitter.Emit('OnOutputPortChanged',pOutputPortChangeEvent^);
pOutputPortChangeEvent^.Dispose();
END_METHOD

METHOD FB_init : BOOL
VAR_INPUT
	bInitRetains : BOOL; // if TRUE, the retain variables are initialized (warm start / cold start)
	bInCopyCode : BOOL;  // if TRUE, the instance afterwards gets moved into the copy code (online change)
	Name : T_MAXSTRING;
	Data : I_Datatype;
	Parent : I_HostOutputPorts;
END_VAR
_name := Name;
_data := Data;
RegisterWithParent(Parent);
END_METHOD

PROPERTY PUBLIC Metadatum : I_Metadatum
GET
Metadatum := metadataHost;
END_GET
END_PROPERTY

PROPERTY PUBLIC Name : T_MAXSTRING
GET
Name := _name;
END_GET
END_PROPERTY

METHOD PUBLIC OffEvent
VAR_INPUT
	EventName : T_MaxString;
	EventHandler : I_EventHandler;
END_VAR
eventEmitter.OffEvent(EventName, EventHandler);
END_METHOD

METHOD PUBLIC OnceEvent
VAR_INPUT
	EventName : T_MaxString;
	EventHandler : I_EventHandler;
END_VAR
eventEmitter.OnceEvent(EventName, EventHandler);
END_METHOD

METHOD PUBLIC OnEvent
VAR_INPUT
	EventName : T_MaxString;
	EventHandler : I_EventHandler;
END_VAR
eventEmitter.OnEvent(EventName, EventHandler);
END_METHOD

METHOD PUBLIC RegisterWithParent
VAR_INPUT
	Parent : I_HostOutputPorts;
END_VAR
IF Parent = 0 THEN
	RETURN;
END_IF

THIS^.parent := Parent;
Parent.OutputPorts.AddOutputPort(THIS^);
END_METHOD

METHOD PUBLIC SerializeWith
VAR_INPUT
	Serializer : I_Serializer;
END_VAR
Serializer.StartObject();
Serializer.AddKeyString('name',_name);
Serializer.Addkey('type');
_data.SerializeTypeWith(Serializer);
Serializer.AddkeyObject('value',_data);
metadataHost.SerializeWith(Serializer);
Serializer.EndObject();
END_METHOD

END_FUNCTION_BLOCK

// ---- OutputPort/Host/OutputPortHost.TcPOU
{attribute 'linkalways'} 
{attribute 'no_explicit_call' := 'This FB is a CLASS and must be accessed using methods or properties'}
{attribute 'enable_dynamic_creation'}
FUNCTION_BLOCK OutputPortHost IMPLEMENTS I_OutputPorts, I_Serializable
VAR
	hostParent : I_HostOutputPorts;
	eventTarget : I_EventTarget;
	ports : OrderedDictionary;
	selfCreatedOutputPorts : Stack;
END_VAR

METHOD PUBLIC Accept
VAR_INPUT
	Visitor : I_OutputPortVisitor;
END_VAR
VAR
	enumerator : I_ForwardEnumerator;
	port : I_OutputPort;
END_VAR
enumerator := ports.GetEnumerator();

WHILE (enumerator.MoveNext()) DO
	
	IF enumerator.TryGet(port) THEN
		port.Accept(Visitor);
	END_IF

END_WHILE

enumerator.Dispose();
END_METHOD

METHOD PUBLIC AddDataAsOutputPort : I_OutputPort
VAR_INPUT
	Name : T_MAXSTRING;
	Data : I_Datatype;
END_VAR
VAR
	port : I_OutputPort;
END_VAR
port := CreateOutputPort(Name, Data);
selfCreatedOutputPorts.Push(port);
AddDataAsOutputPort := port;
END_METHOD

METHOD PUBLIC AddOutputPort
VAR_INPUT
	OutputPort : I_OutputPort;
END_VAR
ports.AddOrUpdate(OutputPort.Name, OutputPort);
EmitOnPortAddedEvent(OutputPort);
END_METHOD

METHOD PRIVATE CreateOutputPort : I_OutputPort
VAR_INPUT
	PortName : T_MAXSTRING;
	PortData : I_Datatype;
END_VAR
VAR
	pPort : POINTER TO OutputPort;
END_VAR
pPort := __NEW(OutputPort(Name := PortName, Data := PortData, Parent := hostParent));
CreateOutputPort := pPort^;
END_METHOD

METHOD PRIVATE DisposeSelfCreatedOutputPorts : BOOL
VAR
	port : I_OutputPort;
END_VAR
WHILE selfCreatedOutputPorts.TryPop(port) DO
	port.Dispose();
END_WHILE
END_METHOD

METHOD PROTECTED EmitOnPortAddedEvent
VAR_INPUT
	Port : I_OutputPort;
END_VAR
VAR
	pOutputPortAddedEvent : POINTER TO OutputPortAddedEvent;
END_VAR
IF eventTarget = 0 THEN
	RETURN;
END_IF

pOutputPortAddedEvent := __NEW(OutputPortAddedEvent(Target := Port));
eventTarget.Emit('OnOutputPortAdded',pOutputPortAddedEvent^);
pOutputPortAddedEvent^.Dispose();
END_METHOD

METHOD FB_exit : BOOL
VAR_INPUT
	bInCopyCode : BOOL; // if TRUE, the exit method is called for exiting an instance that is copied afterwards (online change).
END_VAR
IF bInCopyCode THEN
	RETURN;
END_IF

DisposeSelfCreatedOutputPorts();
END_METHOD

METHOD FB_init : BOOL
VAR_INPUT
	bInitRetains : BOOL; // if TRUE, the retain variables are initialized (warm start / cold start)
	bInCopyCode : BOOL;  // if TRUE, the instance afterwards gets moved into the copy code (online change)
	Parent : I_HostOutputPorts;
	ParentEventTarget : I_EventTarget;
END_VAR
hostParent := Parent;
eventTarget := parentEventTarget;
END_METHOD

PROPERTY PUBLIC HasOutputPorts : BOOL
GET
HasOutputPorts := ports.Count > 0;
END_GET
END_PROPERTY

METHOD PUBLIC SerializeWith
VAR_INPUT
	Serializer : I_Serializer;
END_VAR
VAR
	enumerator : I_ForwardEnumerator;
	port : I_OutputPort;
END_VAR
IF ports.Count = 0 THEN
	RETURN;
END_IF

Serializer.AddKey('outputPorts');
Serializer.StartArray();

enumerator := ports.GetEnumerator();

WHILE enumerator.MoveNext() DO
	IF enumerator.TryGet(port) THEN
		port.SerializeWith(Serializer);
	END_IF
END_WHILE

Serializer.EndArray();
enumerator.Dispose();
END_METHOD

METHOD PUBLIC TryGetOutputPortByName : BOOL
VAR_INPUT
	Name : T_MAXSTRING;
	Destination : REFERENCE TO I_OutputPort;
END_VAR
VAR
	port : I_OutputPort;
END_VAR
IF NOT ports.TryGetValue(Name, port) THEN
	RETURN;
END_IF

Destination := port;
TryGetOutputPortByName := TRUE;
END_METHOD

END_FUNCTION_BLOCK

// ---- Parameters/Host/ParameterHost.TcPOU
{attribute 'linkalways'} 
{attribute 'no_explicit_call' := 'This FB is a CLASS and must be accessed using methods or properties'}
{attribute 'enable_dynamic_creation'}
FUNCTION_BLOCK ParameterHost IMPLEMENTS I_Parameters, I_Serializable
VAR
	hostParent : I_HostParameters;
	eventTarget : I_EventTarget;
	parameters : OrderedDictionary;
	selfCreatedParameters : Stack;
END_VAR

METHOD PUBLIC Accept
VAR_INPUT
	Visitor : I_ParameterVisitor;
END_VAR
VAR
	enumerator : I_ForwardEnumerator;
	parameter : I_Parameter;
END_VAR
enumerator := parameters.GetEnumerator();

WHILE (enumerator.MoveNext()) DO
	
	IF enumerator.TryGet(parameter) THEN
		parameter.Accept(Visitor);
	END_IF

END_WHILE

enumerator.Dispose();
END_METHOD

METHOD PUBLIC AddDataAsParameter : I_Parameter
VAR_INPUT
	Name : T_MAXSTRING;
	Data : I_Datatype;
END_VAR
VAR
	parameter : I_Parameter;
END_VAR
parameter := CreateParameter(Name, Data);
selfCreatedParameters.Push(parameter);
AddDataAsParameter := parameter;
END_METHOD

METHOD PUBLIC AddParameter
VAR_INPUT
	Parameter : I_Parameter;
END_VAR
parameters.AddOrUpdate(Parameter.Name, Parameter);
EmitOnParameterAddedEvent(Parameter);
END_METHOD

METHOD PRIVATE CreateParameter : I_Parameter
VAR_INPUT
	ParameterName : T_MAXSTRING;
	ParameterData : I_Datatype;
END_VAR
VAR
	pParameter : POINTER TO Parameter;
END_VAR
pParameter := __NEW(Parameter(Name := ParameterName, Data := ParameterData, Parent := hostParent));
CreateParameter := pParameter^;
END_METHOD

METHOD PRIVATE DisposeSelfCreatedParameters : BOOL
VAR
	parameter : I_Parameter;
END_VAR
WHILE selfCreatedParameters.TryPop(parameter) DO
	parameter.Dispose();
END_WHILE
END_METHOD

METHOD PROTECTED EmitOnParameterAddedEvent
VAR_INPUT
	Parameter : I_Parameter;
END_VAR
VAR
	pParameterAddedEvent : POINTER TO ParameterAddedEvent;
END_VAR
IF eventTarget = 0 THEN
	RETURN;
END_IF

pParameterAddedEvent := __NEW(ParameterAddedEvent(TargetParameter := Parameter));
eventTarget.Emit('OnParameterAdded',pParameterAddedEvent^);
pParameterAddedEvent^.Dispose();
END_METHOD

METHOD FB_exit : BOOL
VAR_INPUT
	bInCopyCode : BOOL; // if TRUE, the exit method is called for exiting an instance that is copied afterwards (online change).
END_VAR
IF bInCopyCode THEN
	RETURN;
END_IF

DisposeSelfCreatedParameters();
END_METHOD

METHOD FB_init : BOOL
VAR_INPUT
	bInitRetains : BOOL; // if TRUE, the retain variables are initialized (warm start / cold start)
	bInCopyCode : BOOL;  // if TRUE, the instance afterwards gets moved into the copy code (online change)
	Parent : I_HostParameters;
	ParentEventTarget : I_EventTarget;
END_VAR
hostParent := Parent;
eventTarget := ParentEventTarget;
END_METHOD

PROPERTY PUBLIC HasParameters : BOOL
GET
HasParameters := NOT parameters.IsEmpty;
END_GET
END_PROPERTY

METHOD PUBLIC SerializeWith
VAR_INPUT
	Serializer : I_Serializer;
END_VAR
VAR
	enumerator : I_ForwardEnumerator;
	parameter : I_Parameter;
END_VAR
IF parameters.Count = 0 THEN
	RETURN;
END_IF

Serializer.AddKey('parameters');
Serializer.StartArray();

enumerator := parameters.GetEnumerator();

WHILE enumerator.MoveNext() DO
	IF enumerator.TryGet(parameter) THEN
		parameter.SerializeWith(Serializer);
	END_IF
END_WHILE

Serializer.EndArray();
enumerator.Dispose();
END_METHOD

METHOD PUBLIC TryDeserializeFrom : BOOL
VAR_INPUT
	Deserializer : I_Deserializer;
	Feedback : I_DeserializerFeedback;
END_VAR
VAR
	parametersDeserializer : I_Deserializer;
	parametersEnumerator : I_DeserializerObjectForwardEnumerator;
	parameter : I_Parameter;
END_VAR
parametersDeserializer := Deserializer.GetKeyObject('properties');
parametersEnumerator := parametersDeserializer.GetObjectEnumerator();

WHILE parametersEnumerator.MoveNext() DO
	
	IF NOT TryGetParameterByName(parametersEnumerator.Key, parameter) THEN
		CONTINUE;
	END_IF
	
	IF NOT parameter.TryDeserializeFrom(parametersEnumerator.Current, Feedback) THEN
		RETURN;
	END_IF

END_WHILE

TryDeserializeFrom := TRUE;
parametersEnumerator.Dispose();
END_METHOD

METHOD PUBLIC TryGetParameterByName : BOOL
VAR_INPUT
	Name : T_MAXSTRING;
	Destination : REFERENCE TO I_Parameter;
END_VAR
VAR
	parameter : I_Parameter;
END_VAR
IF NOT parameters.TryGetValue(Name, parameter) THEN
	RETURN;
END_IF

Destination := parameter;
TryGetParameterByName := TRUE;
END_METHOD

END_FUNCTION_BLOCK

// ---- Parameters/Base/Parameter.TcPOU
{attribute 'linkalways'} 
{attribute 'no_explicit_call' := 'This FB is a CLASS and must be accessed using methods or properties'}
{attribute 'enable_dynamic_creation'}
FUNCTION_BLOCK Parameter EXTENDS Disposable IMPLEMENTS I_Parameter
VAR
	_name : T_MAXSTRING;
	_data : I_Datatype;
	_parent : I_HostParameters;
	eventEmitter : EventEmitter;
	metadataHost : MetadataHost(THIS^, eventEmitter);
END_VAR

METHOD PUBLIC Accept
VAR_INPUT
	Visitor : I_ParameterVisitor;
END_VAR
Visitor.VisitParameter(THIS^);
END_METHOD

METHOD PUBLIC AddMetadata : I_HostMetadata
VAR_INPUT
	Name : T_MAXSTRING;
	Data : I_Datatype;
END_VAR
Metadatum.AddDataAsMetadata(Name, Data);
AddMetadata := THIS^;
END_METHOD

PROPERTY PUBLIC Data : I_Datatype
GET
Data := _data;
END_GET
END_PROPERTY

METHOD FB_init : BOOL
VAR_INPUT
	bInitRetains : BOOL; // if TRUE, the retain variables are initialized (warm start / cold start)
	bInCopyCode : BOOL;  // if TRUE, the instance afterwards gets moved into the copy code (online change)
	Name : T_MAXSTRING;
	Data : I_Datatype;
	Parent : I_HostParameters;
END_VAR
_name := Name;
_data := Data;
RegisterWithParent(Parent);
END_METHOD

PROPERTY PUBLIC Metadatum : I_Metadatum
GET
Metadatum := metadataHost;
END_GET
END_PROPERTY

PROPERTY PUBLIC Name : T_MAXSTRING
GET
Name := _name;
END_GET
END_PROPERTY

METHOD PUBLIC OffEvent
VAR_INPUT
	EventName : T_MaxString;
	EventHandler : I_EventHandler;
END_VAR
eventEmitter.OffEvent(EventName, EventHandler);
END_METHOD

METHOD PUBLIC OnceEvent
VAR_INPUT
	EventName : T_MaxString;
	EventHandler : I_EventHandler;
END_VAR
eventEmitter.OnceEvent(EventName, EventHandler);
END_METHOD

METHOD PUBLIC OnEvent
VAR_INPUT
	EventName : T_MaxString;
	EventHandler : I_EventHandler;
END_VAR
eventEmitter.OnEvent(EventName, EventHandler);
END_METHOD

PROPERTY PUBLIC Parent : I_HostParameters
GET
Parent := _parent;
END_GET
END_PROPERTY

METHOD PUBLIC RegisterWithParent
VAR_INPUT
	Parent : I_HostParameters;
END_VAR
IF Parent = 0 THEN
	RETURN;
END_IF

THIS^._parent := Parent;
Parent.Parameters.AddParameter(THIS^);
END_METHOD

METHOD PUBLIC SerializeWith
VAR_INPUT
	Serializer : I_Serializer;
END_VAR
Serializer.StartObject();
Serializer.AddKeyString('name',_name);
Serializer.Addkey('type');
_data.SerializeTypeWith(Serializer);
Serializer.AddkeyObject('value',_data);
metadataHost.SerializeWith(Serializer);
Serializer.EndObject();
END_METHOD

METHOD PUBLIC TryDeserializeFrom : BOOL
VAR_INPUT
	Deserializer : I_Deserializer;
	Feedback : I_DeserializerFeedback;
END_VAR
VAR
	parameterDeserializer : I_Deserializer;
END_VAR
TryDeserializeFrom := _data.TryDeserializeFrom(Deserializer, Feedback);
END_METHOD

END_FUNCTION_BLOCK

// ---- Parameters/Events/ParameterAddedEvent.TcPOU
{attribute 'linkalways'} 
{attribute 'no_explicit_call' := 'This FB is a CLASS and must be accessed using methods or properties'}
{attribute 'enable_dynamic_creation'}
FUNCTION_BLOCK ParameterAddedEvent EXTENDS Disposable IMPLEMENTS I_ParameterAddedEvent
VAR
	_targetParameter : I_Parameter;
END_VAR

METHOD FB_init : BOOL
VAR_INPUT
	bInitRetains : BOOL; // if TRUE, the retain variables are initialized (warm start / cold start)
	bInCopyCode : BOOL;  // if TRUE, the instance afterwards gets moved into the copy code (online change)
	TargetParameter : I_Parameter;
END_VAR
This^._targetParameter := TargetParameter;
END_METHOD

PROPERTY PUBLIC TargetParameter : I_Parameter
GET
TargetParameter := _targetParameter;
END_GET
END_PROPERTY

END_FUNCTION_BLOCK

// ---- Content/Host/ContentHost.TcPOU
{attribute 'linkalways'} 
{attribute 'no_explicit_call' := 'This FB is a CLASS and must be accessed using methods or properties'}
{attribute 'enable_dynamic_creation'}
FUNCTION_BLOCK ContentHost IMPLEMENTS I_Contents, I_Serializable
VAR
	hostParent : I_HostContent;
	eventTarget : I_EventTarget;
	contents : OrderedDictionary;
	selfCreatedContent : Stack;
END_VAR

METHOD PUBLIC Accept
VAR_INPUT
	visitor : I_ContentVisitor;
END_VAR
VAR
	enumerator : I_ForwardEnumerator;
	content : I_Content;
END_VAR
enumerator := contents.GetEnumerator();

WHILE (enumerator.MoveNext()) DO
	
	IF enumerator.TryGet(content) THEN
		content.Accept(Visitor);
	END_IF

END_WHILE

enumerator.Dispose();
END_METHOD

METHOD PUBLIC AddContent
VAR_INPUT
	Content : I_Content;
END_VAR
contents.AddOrUpdate(Content.Name, Content);
EmitOnContentAddedEvent(Content);
END_METHOD

METHOD PUBLIC AddDataAsContent : I_Content
VAR_INPUT
	Name : T_MAXSTRING;
	Data : I_Datatype;
END_VAR
VAR
	content : I_Content;
END_VAR
content := CreateContent(Name, Data);
selfCreatedContent.Push(content);
AddDataAsContent := content;
END_METHOD

METHOD PRIVATE CreateContent : I_Content
VAR_INPUT
	ContentName : T_MAXSTRING;
	ContentData : I_Datatype;
END_VAR
VAR
	pContent : POINTER TO Content;
END_VAR
pContent := __NEW(Content(Name := ContentName, Data := ContentData, Parent := hostParent));
CreateContent := pContent^;
END_METHOD

METHOD PRIVATE DisposeSelfCreatedContent : BOOL
VAR
	content : I_Content;
END_VAR
WHILE selfCreatedContent.TryPop(content) DO
	content.Dispose();
END_WHILE
END_METHOD

METHOD PROTECTED EmitOnContentAddedEvent
VAR_INPUT
	Content : I_Content;
END_VAR
VAR
	pContentAddedEvent : POINTER TO ContentAddedEvent;
END_VAR
IF eventTarget = 0 THEN
	RETURN;
END_IF

pContentAddedEvent := __NEW(ContentAddedEvent(Target := Content));
eventTarget.Emit('OnContentAdded',pContentAddedEvent^);
pContentAddedEvent^.Dispose();
END_METHOD

METHOD FB_exit : BOOL
VAR_INPUT
	bInCopyCode : BOOL; // if TRUE, the exit method is called for exiting an instance that is copied afterwards (online change).
END_VAR
IF bInCopyCode THEN
	RETURN;
END_IF

DisposeSelfCreatedContent();
END_METHOD

METHOD FB_init : BOOL
VAR_INPUT
	bInitRetains : BOOL; // if TRUE, the retain variables are initialized (warm start / cold start)
	bInCopyCode : BOOL;  // if TRUE, the instance afterwards gets moved into the copy code (online change)
	Parent : I_HostContent;
	ParentEventTarget : I_EventTarget;
END_VAR
hostParent := Parent;
eventTarget := parentEventTarget;
END_METHOD

PROPERTY PUBLIC HasContents : BOOL
GET
HasContents := NOT contents.IsEmpty;
END_GET
END_PROPERTY

METHOD PUBLIC SerializeWith
VAR_INPUT
	Serializer : I_Serializer;
END_VAR
VAR
	enumerator : I_ForwardEnumerator;
	content : I_Content;
END_VAR
IF contents.Count = 0 THEN
	RETURN;
END_IF

Serializer.AddKey('contents');
Serializer.StartArray();

enumerator := contents.GetEnumerator();

WHILE enumerator.MoveNext() DO
	IF enumerator.TryGet(content) THEN
		content.SerializeWith(Serializer);
	END_IF
END_WHILE

Serializer.EndArray();
enumerator.Dispose();
END_METHOD

METHOD PUBLIC TryGetContentByName : BOOL
VAR_INPUT
	Name : T_MAXSTRING;
	Destination : REFERENCE TO I_Content;
END_VAR
VAR
	content : I_Content;
END_VAR
IF NOT contents.TryGetValue(Name, content) THEN
	RETURN;
END_IF

Destination := content;
TryGetContentByName := TRUE;
END_METHOD

END_FUNCTION_BLOCK

// ---- Content/Base/Content.TcPOU
{attribute 'linkalways'} 
{attribute 'no_explicit_call' := 'This FB is a CLASS and must be accessed using methods or properties'}
{attribute 'enable_dynamic_creation'}
FUNCTION_BLOCK Content EXTENDS Disposable IMPLEMENTS I_Content
VAR
	_name : T_MAXSTRING;
	_data : I_Datatype;
	_parent : I_HostContent;
	eventEmitter : EventEmitter;
	metadataHost : MetadataHost(THIS^, eventEmitter);
END_VAR

METHOD PUBLIC Accept
VAR_INPUT
	Visitor : I_ContentVisitor;
END_VAR
Visitor.VisitContent(THIS^);
END_METHOD

METHOD PUBLIC AddMetadata : I_HostMetadata
VAR_INPUT
	Name : T_MAXSTRING;
	Data : I_Datatype;
END_VAR
Metadatum.AddDataAsMetadata(Name, Data);
AddMetadata := THIS^;
END_METHOD

PROPERTY PUBLIC Data : I_DataType
GET
Data := _data;
END_GET
END_PROPERTY

METHOD FB_init : BOOL
VAR_INPUT
	bInitRetains : BOOL; // if TRUE, the retain variables are initialized (warm start / cold start)
	bInCopyCode : BOOL;  // if TRUE, the instance afterwards gets moved into the copy code (online change)
	Name : T_MAXSTRING;
	Data : I_Datatype;
	Parent : I_HostContent;
END_VAR
_name := Name;
_data := Data;
RegisterWithParent(Parent);
END_METHOD

PROPERTY PUBLIC Metadatum : I_Metadatum
GET
Metadatum := metadataHost;
END_GET
END_PROPERTY

PROPERTY PUBLIC Name : T_MAXSTRING
GET
Name := _name;
END_GET
END_PROPERTY

METHOD PUBLIC OffEvent
VAR_INPUT
	EventName : T_MaxString;
	EventHandler : I_EventHandler;
END_VAR
eventEmitter.OffEvent(EventName, EventHandler);
END_METHOD

METHOD PUBLIC OnceEvent
VAR_INPUT
	EventName : T_MaxString;
	EventHandler : I_EventHandler;
END_VAR
eventEmitter.OnceEvent(EventName, EventHandler);
END_METHOD

METHOD PUBLIC OnEvent
VAR_INPUT
	EventName : T_MaxString;
	EventHandler : I_EventHandler;
END_VAR
eventEmitter.OnEvent(EventName, EventHandler);
END_METHOD

PROPERTY PUBLIC Parent : I_HostContent
GET
Parent := _parent;
END_GET
END_PROPERTY

METHOD PUBLIC RegisterWithParent
VAR_INPUT
	Parent : I_HostContent;
END_VAR
IF Parent = 0 THEN
	RETURN;
END_IF

THIS^._parent := Parent;
Parent.Contents.AddContent(THIS^);
END_METHOD

METHOD PUBLIC SerializeWith
VAR_INPUT
	Serializer : I_Serializer;
END_VAR
Serializer.StartObject();
Serializer.AddKeyString('name',_name);
Serializer.Addkey('datatype');
_data.SerializeTypeWith(Serializer);
Serializer.AddkeyObject('value',_data);
metadataHost.SerializeWith(Serializer);
Serializer.EndObject();
END_METHOD

END_FUNCTION_BLOCK

// ---- Alarms/Host/AlarmHost.TcPOU
{attribute 'linkalways'} 
{attribute 'no_explicit_call' := 'This FB is a CLASS and must be accessed using methods or properties'}
{attribute 'enable_dynamic_creation'}
FUNCTION_BLOCK AlarmHost IMPLEMENTS I_Alarms, I_Serializable
VAR
	hostParent : I_HostAlarms;
	eventTarget : I_EventTarget;
	alarms : Stack;
END_VAR

METHOD PUBLIC Accept
VAR_INPUT
	Visitor : I_AlarmVisitor;
END_VAR
VAR
	enumerator : I_ForwardEnumerator;
	alarm : I_Alarm;
END_VAR
enumerator := alarms.GetEnumerator();

WHILE (enumerator.MoveNext()) DO
	
	IF enumerator.TryGet(alarm) THEN
		alarm.Accept(Visitor);
	END_IF

END_WHILE

enumerator.Dispose();
END_METHOD

METHOD PUBLIC AddAlarm
VAR_INPUT
	Alarm : I_Alarm;
END_VAR
alarms.Push(Alarm);
EmitOnAlarmAddedEvent(Alarm);
END_METHOD

METHOD PROTECTED EmitOnAlarmAddedEvent
VAR_INPUT
	Alarm : I_Alarm;
END_VAR
VAR
	pAlarmAddedEvent : POINTER TO AlarmAddedEvent;
END_VAR
IF eventTarget = 0 THEN
	RETURN;
END_IF

pAlarmAddedEvent := __NEW(AlarmAddedEvent(Target := Alarm));
eventTarget.Emit('OnAlarmAdded',pAlarmAddedEvent^);
pAlarmAddedEvent^.Dispose();
END_METHOD

METHOD FB_init : BOOL
VAR_INPUT
	bInitRetains : BOOL; // if TRUE, the retain variables are initialized (warm start / cold start)
	bInCopyCode : BOOL;  // if TRUE, the instance afterwards gets moved into the copy code (online change)
	Parent : I_HostAlarms;
	ParentEventTarget : I_EventTarget;
END_VAR
hostParent := Parent;
eventTarget := parentEventTarget;
END_METHOD

PROPERTY PUBLIC HasAlarms : BOOL
GET
HasAlarms := alarms.Count > 0;
END_GET
END_PROPERTY

PROPERTY PUBLIC HasRaisedAlarm : BOOL
GET
VAR
	enumerator : I_ForwardEnumerator;
	alarm : I_Alarm;
END_VAR
enumerator := alarms.GetEnumerator();

WHILE (enumerator.MoveNext()) DO
	
	IF NOT enumerator.TryGet(alarm) THEN
		CONTINUE;
	END_IF
	
	IF alarm.Active THEN
		HasRaisedAlarm := TRUE;
		EXIT;
	END_IF

END_WHILE

enumerator.Dispose();
END_GET
END_PROPERTY

METHOD PUBLIC SerializeWith
VAR_INPUT
	Serializer : I_Serializer;
END_VAR
VAR
	enumerator : I_ForwardEnumerator;
	alarm : I_Alarm;
END_VAR
IF alarms.Count = 0 THEN
	RETURN;
END_IF

Serializer.AddKey('alarms');
Serializer.StartArray();

enumerator := alarms.GetEnumerator();

WHILE enumerator.MoveNext() DO
	IF enumerator.TryGet(alarm) THEN
		alarm.SerializeWith(Serializer);
	END_IF
END_WHILE

Serializer.EndArray();
enumerator.Dispose();
END_METHOD

END_FUNCTION_BLOCK

// ---- Extensions/Host/ExtensionHost.TcPOU
{attribute 'linkalways'} 
{attribute 'no_explicit_call' := 'This FB is a CLASS and must be accessed using methods or properties'}
{attribute 'enable_dynamic_creation'}
FUNCTION_BLOCK ExtensionHost IMPLEMENTS I_Extensions, I_Serializable, I_Deserializable
VAR
	hostParent : I_HostExtensions;
	eventTarget : I_EventTarget;
	extensions : OrderedDictionary;
END_VAR

METHOD PUBLIC Accept
VAR_INPUT
	Visitor : I_ExtensionVisitor;
END_VAR
VAR
	enumerator : I_ForwardEnumerator;
	extension : I_Extension;
END_VAR
enumerator := extensions.GetEnumerator();

WHILE (enumerator.MoveNext()) DO
	
	IF enumerator.TryGet(extension) THEN
		extension.Accept(Visitor);
	END_IF

END_WHILE

enumerator.Dispose();
END_METHOD

METHOD PUBLIC AddExtension
VAR_INPUT
	Extension : I_Extension;
END_VAR
extensions.AddOrUpdate(Extension.Name,Extension);
EmitOnExtensionAddedEvent(Extension);
END_METHOD

METHOD PROTECTED EmitOnExtensionAddedEvent
VAR_INPUT
	Extension : I_Extension;
END_VAR
VAR
	pExtensionAddedEvent : POINTER TO ExtensionAddedEvent;
END_VAR
IF eventTarget = 0 THEN
	RETURN;
END_IF

pExtensionAddedEvent := __NEW(ExtensionAddedEvent(Target := Extension));
eventTarget.Emit('OnExtensionAdded',pExtensionAddedEvent^);
pExtensionAddedEvent^.Dispose();
END_METHOD

METHOD FB_init : BOOL
VAR_INPUT
	bInitRetains : BOOL; // if TRUE, the retain variables are initialized (warm start / cold start)
	bInCopyCode : BOOL;  // if TRUE, the instance afterwards gets moved into the copy code (online change)
	Parent : I_HostExtensions;
	ParentEventTarget : I_EventTarget;
END_VAR
hostParent := Parent;
eventTarget := parentEventTarget;
END_METHOD

PROPERTY PUBLIC HasExtensions : BOOL
GET
HasExtensions := extensions.Count > 0;
END_GET
END_PROPERTY

METHOD PUBLIC SerializeWith
VAR_INPUT
	Serializer : I_Serializer;
END_VAR
VAR
	enumerator : I_ForwardEnumerator;
	extension : I_Extension;
END_VAR
IF extensions.Count = 0 THEN
	RETURN;
END_IF

Serializer.AddKey('extensions');
Serializer.StartArray();

enumerator := extensions.GetEnumerator();

WHILE enumerator.MoveNext() DO
	IF enumerator.TryGet(extension) THEN
		extension.SerializeWith(Serializer);
	END_IF
END_WHILE

Serializer.EndArray();
enumerator.Dispose();
END_METHOD

METHOD public TryDeserializeFrom : BOOL
VAR_INPUT
	Deserializer : I_Deserializer;
	Feedback : I_DeserializerFeedback;
END_VAR
VAR
	extensionsDeserializer : I_Deserializer;
	extensionsEnumerator : I_DeserializerArrayForwardEnumerator;
	extensionName : T_MAXSTRING;
	extension : I_Extension;
END_VAR
extensionsDeserializer := Deserializer.GetKeyArray('extensions');
extensionsEnumerator := extensionsDeserializer.GetArrayEnumerator();

WHILE extensionsEnumerator.MoveNext() DO
	
	IF NOT extensionsEnumerator.Current.TryGetKeyString('name', extensionName, Feedback) THEN
		CONTINUE;
	END_IF
	
	IF NOT TryGetExtensionByName(extensionName, extension) THEN
		CONTINUE;
	END_IF
	
	IF NOT extension.TryDeserializeFrom(extensionsEnumerator.Current, Feedback) THEN
		extensionsEnumerator.Dispose();
		RETURN;
	END_IF

END_WHILE

TryDeserializeFrom := TRUE;
extensionsEnumerator.Dispose();
END_METHOD

METHOD PUBLIC TryGetExtensionByName : BOOL
VAR_INPUT
	Name : T_MAXSTRING;
	Destination : REFERENCE TO I_Extension;
END_VAR
VAR
	extension : I_Extension;
END_VAR
IF NOT extensions.TryGetValue(Name, extension) THEN
	RETURN;
END_IF

Destination := extension;
TryGetExtensionByName := TRUE;
END_METHOD

END_FUNCTION_BLOCK

// ---- Extensions/Base/Extension.TcPOU
{attribute 'linkalways'} 
{attribute 'no_explicit_call' := 'This FB is a CLASS and must be accessed using methods or properties'}
{attribute 'enable_dynamic_creation'}
{attribute 'hide_all_locals'}
FUNCTION_BLOCK Extension EXTENDS Disposable IMPLEMENTS I_Extension
VAR
	_name : T_MAXSTRING;
	_parent : I_HostExtensions;
	eventEmitter : EventEmitter;
	inputPortHost : InputPortHost(THIS^, eventEmitter);
	outputPortHost : OutputPortHost(THIS^, eventEmitter);
	parameterHost : ParameterHost(THIS^, eventEmitter);
	contentHost : ContentHost(THIS^, eventEmitter);
	alarmHost : AlarmHost(THIS^, eventEmitter);
	metadataHost : MetadataHost(THIS^, eventEmitter);
	deserializationFailedAlarm : DeserializationFailedAlarm(THIS^);
END_VAR

METHOD PUBLIC Accept
VAR_INPUT
	Visitor : I_ExtensionVisitor;
END_VAR
Visitor.VisitExtension(THIS^);
END_METHOD

METHOD PROTECTED AddContent : I_Content
VAR_INPUT
	Name : T_MAXSTRING;
	Data : I_Datatype;
END_VAR
AddContent := Contents.AddDataAsContent(Name, Data);
END_METHOD

METHOD PROTECTED AddInput : I_InputPort
VAR_INPUT
	Name : T_MAXSTRING;
	Data : I_Datatype;
END_VAR
AddInput := InputPorts.AddDataAsInputPort(Name, Data);
END_METHOD

METHOD PUBLIC AddMetadata : I_HostMetadata
VAR_INPUT
	Name : T_MAXSTRING;
	Data : I_Datatype;
END_VAR
Metadatum.AddDataAsMetadata(Name, Data);
AddMetadata := THIS^;
END_METHOD

METHOD PROTECTED AddOutput : I_OutputPort
VAR_INPUT
	Name : T_MAXSTRING;
	Data : I_Datatype;
END_VAR
AddOutput := OutputPorts.AddDataAsOutputPort(Name, Data);
END_METHOD

METHOD PROTECTED AddParameter : I_Parameter
VAR_INPUT
	Name : T_MAXSTRING;
	Data : I_Datatype;
END_VAR
AddParameter := Parameters.AddDataAsParameter(Name, Data);
END_METHOD

PROPERTY PUBLIC Alarms : I_Alarms
GET
Alarms := alarmHost;
END_GET
END_PROPERTY

PROPERTY PUBLIC Contents : I_Contents
GET
Contents := contentHost;
END_GET
END_PROPERTY

METHOD FB_init : BOOL
VAR_INPUT
	bInitRetains : BOOL; // if TRUE, the retain variables are initialized (warm start / cold start)
	bInCopyCode : BOOL;  // if TRUE, the instance afterwards gets moved into the copy code (online change)
	Name : T_MAXSTRING;
	Parent : I_HostExtensions;
END_VAR
_name := Name;
RegisterWithParent(Parent);
END_METHOD

PROPERTY PUBLIC HasRaisedAlarm : BOOL
GET
HasRaisedAlarm := alarmHost.HasRaisedAlarm;
END_GET
END_PROPERTY

PROPERTY PUBLIC InputPorts : I_InputPorts
GET
InputPorts := inputPortHost;
END_GET
END_PROPERTY

PROPERTY PUBLIC Metadatum : I_Metadatum
GET
Metadatum := metadataHost;
END_GET
END_PROPERTY

PROPERTY PUBLIC Name : T_MAXSTRING
GET
Name := _name;
END_GET
END_PROPERTY

METHOD PUBLIC OffEvent
VAR_INPUT
	EventName : T_MaxString;
	EventHandler : I_EventHandler;
END_VAR
eventEmitter.OffEvent(EventName, EventHandler);
END_METHOD

METHOD PUBLIC OnceEvent
VAR_INPUT
	EventName : T_MaxString;
	EventHandler : I_EventHandler;
END_VAR
eventEmitter.OnceEvent(EventName, EventHandler);
END_METHOD

METHOD PUBLIC OnEvent
VAR_INPUT
	EventName : T_MaxString;
	EventHandler : I_EventHandler;
END_VAR
eventEmitter.OnEvent(EventName, EventHandler);
END_METHOD

PROPERTY PUBLIC OutputPorts : I_OutputPorts
GET
OutputPorts := outputPortHost;
END_GET
END_PROPERTY

PROPERTY PUBLIC Parameters : I_Parameters
GET
Parameters := parameterHost;
END_GET
END_PROPERTY

PROPERTY PUBLIC Parent : I_HostExtensions
GET
Parent := _parent;
END_GET
END_PROPERTY

METHOD PUBLIC RegisterWithParent
VAR_INPUT
	Parent : I_HostExtensions;
END_VAR
IF Parent = 0 THEN
	RETURN;
END_IF

_parent := Parent;
Parent.Extensions.AddExtension(THIS^);
END_METHOD

METHOD PUBLIC SerializeWith
VAR_INPUT
	Serializer : I_Serializer;
END_VAR
Serializer.StartObject();
Serializer.AddKeyString('name',_name);
inputPortHost.SerializeWith(Serializer);
outputPortHost.SerializeWith(Serializer);
parameterHost.SerializeWith(Serializer);
contentHost.SerializeWith(Serializer);
alarmHost.SerializeWith(Serializer);
metadataHost.SerializeWith(Serializer);
Serializer.EndObject();
END_METHOD

METHOD PUBLIC TryDeserializeFrom : BOOL
VAR_INPUT
	Deserializer : I_Deserializer;
	Feedback : I_DeserializerFeedback;
END_VAR
DeserializationFailedAlarm.Clear();

IF NOT parameterHost.TryDeserializeFrom(Deserializer, Feedback) THEN
	DeserializationFailedAlarm.Raise('Failed to deserialize parameters');
	RETURN;
END_IF

TryDeserializeFrom := TRUE;
END_METHOD

END_FUNCTION_BLOCK

// ---- Extensions/Events/ExtensionAddedEvent.TcPOU
{attribute 'linkalways'} 
{attribute 'no_explicit_call' := 'This FB is a CLASS and must be accessed using methods or properties'}
{attribute 'enable_dynamic_creation'}
FUNCTION_BLOCK ExtensionAddedEvent EXTENDS Disposable IMPLEMENTS I_ExtensionAddedEvent
VAR
	_target : I_Extension;
END_VAR

METHOD FB_init : BOOL
VAR_INPUT
	bInitRetains : BOOL; // if TRUE, the retain variables are initialized (warm start / cold start)
	bInCopyCode : BOOL;  // if TRUE, the instance afterwards gets moved into the copy code (online change)
	Target : I_Extension;
END_VAR
This^._target := Target;
END_METHOD

PROPERTY PUBLIC Target : I_Extension
GET
Target := _target;
END_GET
END_PROPERTY

END_FUNCTION_BLOCK

// ---- Node/Events/NodeExecuteBeginEvent.TcPOU
{attribute 'linkalways'} 
{attribute 'no_explicit_call' := 'This FB is a CLASS and must be accessed using methods or properties'}
{attribute 'enable_dynamic_creation'}
FUNCTION_BLOCK NodeExecuteBeginEvent EXTENDS Disposable IMPLEMENTS I_NodeExecuteBeginEvent
VAR
	_target : I_Node;
	_cpuCounterLowBytes : UDINT;
	_cpuCounterHighBytes : UDINT;
END_VAR

PROPERTY PUBLIC CpuCounterHighBytes : UDINT
GET
CpuCounterHighBytes := _cpuCounterHighBytes;
END_GET
END_PROPERTY

PROPERTY PUBLIC CpuCounterLowBytes : UDINT
GET
CpuCounterLowBytes := _cpuCounterLowBytes;
END_GET
END_PROPERTY

METHOD FB_init : BOOL
VAR_INPUT
	bInitRetains : BOOL; // if TRUE, the retain variables are initialized (warm start / cold start)
	bInCopyCode : BOOL;  // if TRUE, the instance afterwards gets moved into the copy code (online change)
	Target : I_Node;
END_VAR
VAR
	getCount : GETCPUCOUNTER;
END_VAR
_target := Target;
getCount(cpuCntLoDW => _cpuCounterLowBytes, cpuCntHiDW => _cpuCounterHighBytes);
END_METHOD

PROPERTY PUBLIC Target : I_Node
GET
Target := _target;
END_GET
END_PROPERTY

END_FUNCTION_BLOCK

// ---- Node/Events/NodeExecuteEndEvent.TcPOU
{attribute 'linkalways'} 
{attribute 'no_explicit_call' := 'This FB is a CLASS and must be accessed using methods or properties'}
{attribute 'enable_dynamic_creation'}
FUNCTION_BLOCK NodeExecuteEndEvent EXTENDS Disposable IMPLEMENTS I_NodeExecuteEndEvent
VAR
	_target : I_Node;
	_cpuCounterLowBytes : UDINT;
	_cpuCounterHighBytes : UDINT;
END_VAR

PROPERTY PUBLIC CpuCounterHighBytes : UDINT
GET
CpuCounterHighBytes := _cpuCounterHighBytes;
END_GET
END_PROPERTY

PROPERTY PUBLIC CpuCounterLowBytes : UDINT
GET
CpuCounterLowBytes := _cpuCounterLowBytes;
END_GET
END_PROPERTY

METHOD FB_init : BOOL
VAR_INPUT
	bInitRetains : BOOL; // if TRUE, the retain variables are initialized (warm start / cold start)
	bInCopyCode : BOOL;  // if TRUE, the instance afterwards gets moved into the copy code (online change)
	Target : I_Node;
END_VAR
VAR
	getCount : GETCPUCOUNTER;
END_VAR
_target := Target;
getCount(cpuCntLoDW => _cpuCounterLowBytes, cpuCntHiDW => _cpuCounterHighBytes);
END_METHOD

PROPERTY PUBLIC Target : I_Node
GET
Target := _target;
END_GET
END_PROPERTY

END_FUNCTION_BLOCK

// ---- Node/Events/NodePreExecuteEvent.TcPOU
{attribute 'linkalways'} 
{attribute 'no_explicit_call' := 'This FB is a CLASS and must be accessed using methods or properties'}
{attribute 'enable_dynamic_creation'}
FUNCTION_BLOCK NodePreExecuteEvent EXTENDS Disposable IMPLEMENTS I_NodePreExecuteEvent
VAR
	_target : I_Node;
	_cancelExecute : BOOL;
END_VAR

METHOD PUBLIC Cancel
VAR_INPUT
END_VAR
_cancelExecute := true;
END_METHOD

PROPERTY PUBLIC ExecuteCancelled : BOOL
GET
ExecuteCancelled := _cancelExecute;
END_GET
END_PROPERTY

METHOD FB_init : BOOL
VAR_INPUT
	bInitRetains : BOOL; // if TRUE, the retain variables are initialized (warm start / cold start)
	bInCopyCode : BOOL;  // if TRUE, the instance afterwards gets moved into the copy code (online change)
	Target : I_Node;
END_VAR
_target := Target;
END_METHOD

METHOD PUBLIC Reinitialize
VAR_INPUT
	Target : I_Node;
END_VAR
_cancelExecute := FALSE;
_target := Target;
END_METHOD

PROPERTY PUBLIC Target : I_Node
GET
Target := _target;
END_GET
END_PROPERTY

END_FUNCTION_BLOCK

// ---- Alarms/FunctionFailedAlarm.TcPOU
{attribute 'linkalways'} 
{attribute 'no_explicit_call' := 'This FB is a CLASS and must be accessed using methods or properties'}
{attribute 'enable_dynamic_creation'}
FUNCTION_BLOCK PUBLIC FunctionFailedAlarm EXTENDS Alarm
VAR
	state : (CLEARED, RAISED);
	functionName : STRING;
	hresult : HRESULT;
END_VAR

PROPERTY Active : BOOL
GET
Active := state <> CLEARED;
END_GET
END_PROPERTY

METHOD PUBLIC Clear
functionName := '';
hresult := 0;
state := CLEARED;
END_METHOD

PROPERTY Message : T_MaxString
GET
Message := 'Function failed';
END_GET
END_PROPERTY

METHOD PUBLIC Raise
VAR_INPUT
	FunctionName : STRING;
	HResult : HRESULT;
END_VAR
THIS^.functionName := FunctionName;
THIS^.hresult := HResult;
state := RAISED;
END_METHOD

PROPERTY Reason : T_MaxString
GET
VAR
	message : STRING;
	returnCode : DWORD;
	returnCodeString : STRING;
	returnCodeMsg : STRING;
END_VAR
IF state = CLEARED THEN
	RETURN;
END_IF

returnCode := DINT_TO_DWORD(hresult) AND 16#FFF;
returnCodeString := DWORD_TO_HEXSTR(returnCode, 3, FALSE);

CASE (returnCode) OF
	
	16#70A: returnCodeMsg := 'NOMEMORY';
	16#70B: returnCodeMsg := 'INVALIDPARM';
	16#70C: returnCodeMsg := 'NOTFOUND';
	16#70E: returnCodeMsg := 'INCOMPATIBLE';
	16#712: returnCodeMsg := 'INVALIDSTATE';
	16#719: returnCodeMsg := 'TIMEOUT';
	16#71A: returnCodeMsg := 'NOINTERFACE';
	16#71B: returnCodeMsg := 'INVALIDINTERFACE';
	16#71D: returnCodeMsg := 'INVALIDOBJID';
	16#734: returnCodeMsg := 'OUTOFRANGE';
	
END_CASE


message := functionName;
message := CONCAT(message,', Msg : ');
message := CONCAT(message,returnCodeMsg);
message := CONCAT(message,', Code : 16#');
message := CONCAT(message,returnCodeString);

Reason := message;
END_GET
END_PROPERTY

END_FUNCTION_BLOCK

// ---- API/GraphFrameworkApi.TcPOU
{attribute 'linkalways'} 
{attribute 'no_explicit_call' := 'This FB is a CLASS and must be accessed using methods or properties'}
{attribute 'enable_dynamic_creation'}
FUNCTION_BLOCK GraphFrameworkApi IMPLEMENTS I_RpcApi, I_HostGraphs, I_EventEmitter
VAR
	graphFramework : I_GraphFramework;
	eventEmitter : EventEmitter;
	graphHost : GraphHost(THIS^, eventEmitter);
	createGraphRpcHandler : CreateGraphRpcHandler;
	createGraphMultiUserRpcHandler : CreateGraphMultiUserRpcHandler;
	getStatusRpcHandler : GetStatusRpcHandler;
	getBlueprintsRpcHandler : GetBlueprintsRpcHandler;
	getContentValueHandler : GetContentValueHandler;
	updateParameterValueHandler : UpdateParameterValueHandler;
END_VAR

METHOD PUBLIC CyclicCall
VAR_INPUT
END_VAR
graphHost.Execute();
END_METHOD

METHOD FB_exit : BOOL
VAR_INPUT
	bInCopyCode : BOOL; // if TRUE, the exit method is called for exiting an instance that is copied afterwards (online change).
END_VAR
IF bInCopyCode THEN
	RETURN;
END_IF

graphs.DisposeAll();
END_METHOD

METHOD FB_init : BOOL
VAR_INPUT
	bInitRetains : BOOL; // if TRUE, the retain variables are initialized (warm start / cold start)
	bInCopyCode : BOOL;  // if TRUE, the instance afterwards gets moved into the copy code (online change)
	GraphFramework : I_GraphFramework;
END_VAR
THIS^.graphFramework := GraphFramework;

getBlueprintsRpcHandler.Initialize(GraphFramework.NodeFactory);
getStatusRpcHandler.Initialize(graphHost);
createGraphRpcHandler.Initialize(GraphFramework, graphHost);
createGraphMultiUserRpcHandler.Initialize(GraphFramework, graphHost);
getContentValueHandler.Initialize(graphHost);
updateParameterValueHandler.Initialize(graphHost);
END_METHOD

PROPERTY PUBLIC Graphs : I_Graphs
GET
Graphs := graphHost;
END_GET
END_PROPERTY

METHOD PUBLIC OffEvent
VAR_INPUT
	EventName : T_MaxString;
	EventHandler : I_EventHandler;
END_VAR
eventEmitter.OffEvent(EventName, EventHandler);
END_METHOD

METHOD PUBLIC OnceEvent
VAR_INPUT
	EventName : T_MaxString;
	EventHandler : I_EventHandler;
END_VAR
eventEmitter.OnceEvent(EventName, EventHandler);
END_METHOD

METHOD PUBLIC OnEvent
VAR_INPUT
	EventName : T_MaxString;
	EventHandler : I_EventHandler;
END_VAR
eventEmitter.OnEvent(EventName, EventHandler);
END_METHOD

METHOD RegisterAsynchronousRpcHandlersWith
VAR_INPUT
	Host : I_HostAsynchronousRpcHandlers;
END_VAR
Host.RegisterHandler('CreateGraph',createGraphRpcHandler);
Host.RegisterHandler('CreateGraphMultiUser',createGraphMultiUserRpcHandler);
Host.RegisterHandler('GetStatus',getStatusRpcHandler);
Host.RegisterHandler('GetBlueprints',getBlueprintsRpcHandler);
Host.RegisterHandler('GetContentValue',getContentValueHandler);
Host.RegisterHandler('UpdateParameterValue',updateParameterValueHandler);
END_METHOD

METHOD RegisterSynchronousRpcHandlersWith
VAR_INPUT
	Host : I_HostSynchronousRpcHandlers;
END_VAR
// no implementation
END_METHOD

END_FUNCTION_BLOCK

// ---- GraphFramework/GraphFramework.TcPOU
{attribute 'linkalways'} 
{attribute 'no_explicit_call' := 'This FB is a CLASS and must be accessed using methods or properties'}
{attribute 'enable_dynamic_creation'}
FUNCTION_BLOCK GraphFramework IMPLEMENTS I_GraphFramework
VAR
	_nodeFactory : NodeFactory;
	_datatypes : Datatypes;
	datatypeNodeFactory : DatatypeNodeFactory(_datatypes,_nodeFactory);
END_VAR

METHOD PUBLIC Create : I_Graph
VAR
	pGraph : POINTER TO Graph;
END_VAR
pGraph := __NEW(Graph(NodeFactory := _nodeFactory));
Create := pGraph^;
END_METHOD

PROPERTY PUBLIC Datatypes : I_Datatypes
GET
Datatypes := _datatypes;
END_GET
END_PROPERTY

METHOD PUBLIC Install
VAR_INPUT
	Pack : I_GraphPack;
END_VAR
Pack.RegisterWithDatatypes(Datatypes);
Pack.RegisterWithNodeFactory(NodeFactory);
END_METHOD

PROPERTY PUBLIC NodeFactory : I_NodeFactory
GET
NodeFactory := _nodeFactory;
END_GET
END_PROPERTY

END_FUNCTION_BLOCK

// ---- NodeFactory/Base/NodeFactory.TcPOU
{attribute 'linkalways'} 
{attribute 'no_explicit_call' := 'This FB is a CLASS and must be accessed using methods or properties'}
{attribute 'enable_dynamic_creation'}
FUNCTION_BLOCK NodeFactory IMPLEMENTS I_NodeFactory
VAR
	prototypeHost : NodePrototypeHost;
END_VAR

METHOD PUBLIC Accept
VAR_INPUT
	Visitor : I_NodeFactoryVisitor;
END_VAR
Visitor.VisitNodeFactory(this^);
END_METHOD

METHOD AddNodeAsPrototype : I_NodePrototype
VAR_INPUT
	Path : T_MAXSTRING;
	Node : I_Node;
END_VAR
AddNodeAsPrototype := prototypeHost.AddNodeAsPrototype(Path, Node);
END_METHOD

METHOD PUBLIC AddNodePrototype
VAR_INPUT
	NodePrototype : I_NodePrototype;
END_VAR
prototypeHost.AddNodePrototype(NodePrototype);
END_METHOD

PROPERTY PUBLIC NodePrototypes : I_NodePrototypes
GET
NodePrototypes := prototypeHost;
END_GET
END_PROPERTY

METHOD PUBLIC TryCreateNodeByType : BOOL
VAR_INPUT
	Path : T_MAXSTRING;
	Destination : REFERENCE TO I_Node;
END_VAR
VAR
	nodePrototype : I_NodePrototype;
END_VAR
IF NOT prototypeHost.TryGetNodePrototypeByPath(Path, nodePrototype) THEN
	RETURN;
END_IF

Destination := nodePrototype.Clone();
TryCreateNodeByType := TRUE;
END_METHOD

END_FUNCTION_BLOCK

// ---- NodePrototype/Host/NodePrototypeHost.TcPOU
{attribute 'linkalways'} 
{attribute 'no_explicit_call' := 'This FB is a CLASS and must be accessed using methods or properties'}
{attribute 'enable_dynamic_creation'}
FUNCTION_BLOCK NodePrototypeHost IMPLEMENTS I_NodePrototypes
VAR
	prototypes : OrderedDictionary;
	selfCreatedPrototypes : Stack;
END_VAR

METHOD PUBLIC Accept
VAR_INPUT
	visitor : I_NodePrototypeVisitor;
END_VAR
VAR
	enumerator : I_ForwardEnumerator;
	nodePrototype : I_NodePrototype;
END_VAR
enumerator := prototypes.GetEnumerator();

WHILE enumerator.MoveNext() DO
	
	IF enumerator.TryGet(nodePrototype) THEN
		nodePrototype.Accept(Visitor);
	END_IF

END_WHILE

enumerator.Dispose();
END_METHOD

METHOD AddNodeAsPrototype : I_NodePrototype
VAR_INPUT
	Path : T_MAXSTRING;
	Node : I_Node;
END_VAR
VAR
	prototype : I_NodePrototype;
END_VAR
prototype := CreatePrototype(Path, Node);
selfCreatedPrototypes.Push(prototype);
AddNodePrototype(prototype);
AddNodeAsPrototype := prototype;
END_METHOD

METHOD PUBLIC AddNodePrototype
VAR_INPUT
	NodePrototype : I_NodePrototype;
END_VAR
prototypes.AddOrUpdate(NodePrototype.Path, NodePrototype);
END_METHOD

METHOD PRIVATE CreatePrototype : I_NodePrototype
VAR_INPUT
	PrototypePath : T_MAXSTRING;
	PrototypeNode : I_Node;
END_VAR
VAR
	pNodePrototype : POINTER TO NodePrototype;
END_VAR
pNodePrototype := __NEW(NodePrototype(Path := PrototypePath, Node := PrototypeNode));
CreatePrototype := pNodePrototype^;
END_METHOD

METHOD PRIVATE DisposeSelfCreatedNodePrototypes : BOOL
VAR
	prototype : I_NodePrototype;
END_VAR
WHILE selfCreatedPrototypes.TryPop(prototype) DO
	prototype.Dispose();
END_WHILE
END_METHOD

METHOD FB_exit : BOOL
VAR_INPUT
	bInCopyCode : BOOL; // if TRUE, the exit method is called for exiting an instance that is copied afterwards (online change).
END_VAR
IF bInCopyCode THEN
	RETURN;
END_IF

DisposeSelfCreatedNodePrototypes();
END_METHOD

PROPERTY PUBLIC HasNodePrototypes : BOOL
GET
HasNodePrototypes := NOT prototypes.IsEmpty;
END_GET
END_PROPERTY

METHOD PUBLIC TryGetNodePrototypeByPath : BOOL
VAR_INPUT
	Path : T_MAXSTRING;
	Destination : REFERENCE TO I_NodePrototype;
END_VAR
VAR
	nodePrototype : I_NodePrototype;
END_VAR
IF NOT prototypes.TryGetValue(Path, nodePrototype) THEN
	RETURN;
END_IF

Destination := nodePrototype;
TryGetNodePrototypeByPath := TRUE;
END_METHOD

END_FUNCTION_BLOCK

// ---- NodeFactory/Datatype/DatatypeNodeFactory.TcPOU
{attribute 'linkalways'} 
{attribute 'no_explicit_call' := 'This FB is a CLASS and must be accessed using methods or properties'}
{attribute 'enable_dynamic_creation'}
FUNCTION_BLOCK DatatypeNodeFactory IMPLEMENTS I_EventHandler
VAR
	datatypes : I_Datatypes;
	nodeFactory : I_NodeFactory;
	selfCreatedNodes : Stack;
END_VAR

METHOD PROTECTED CreateAliasArrayBundleNode : I_Node
VAR_INPUT
	NodeDatatype : I_AliasDatatype;
END_VAR
VAR
	pAnyBundleNode : POINTER TO AnyAliasArrayBundleNode;
END_VAR
pAnyBundleNode := __NEW(AnyAliasArrayBundleNode(AliasDatatype := NodeDatatype));
CreateAliasArrayBundleNode := pAnyBundleNode^;
END_METHOD

METHOD PROTECTED CreateAliasArrayUnbundleNode : I_Node
VAR_INPUT
	NodeDatatype : I_AliasDatatype;
END_VAR
VAR
	pAnyUnbundleNode : POINTER TO AnyAliasArrayUnbundleNode;
END_VAR
pAnyUnbundleNode := __NEW(AnyAliasArrayUnbundleNode(AliasDatatype := NodeDatatype));
CreateAliasArrayUnbundleNode := pAnyUnbundleNode^;
END_METHOD

METHOD PROTECTED CreateAliasStructureBundleNode : I_Node
VAR_INPUT
	NodeDatatype : I_AliasDatatype;
END_VAR
VAR
	pAnyBundleNode : POINTER TO AnyAliasStructureBundleNode;
END_VAR
pAnyBundleNode := __NEW(AnyAliasStructureBundleNode(AliasDatatype := NodeDatatype));
CreateAliasStructureBundleNode := pAnyBundleNode^;
END_METHOD

METHOD PROTECTED CreateAliasStructureUnbundleNode : I_Node
VAR_INPUT
	NodeDatatype : I_AliasDatatype;
END_VAR
VAR
	pAnyUnbundleNode : POINTER TO AnyAliasStructureUnbundleNode;
END_VAR
pAnyUnbundleNode := __NEW(AnyAliasStructureUnbundleNode(AliasDatatype := NodeDatatype));
CreateAliasStructureUnbundleNode := pAnyUnbundleNode^;
END_METHOD

METHOD PROTECTED CreateArrayBundleNode : I_Node
VAR_INPUT
	NodeDatatype : I_ArrayDatatype;
END_VAR
VAR
	pAnyBundleNode : POINTER TO AnyArrayBundleNode;
END_VAR
pAnyBundleNode := __NEW(AnyArrayBundleNode(ArrayDatatype := NodeDatatype));
CreateArrayBundleNode := pAnyBundleNode^;
END_METHOD

METHOD PROTECTED CreateArrayUnbundleNode : I_Node
VAR_INPUT
	NodeDatatype : I_ArrayDatatype;
END_VAR
VAR
	pAnyUnbundleNode : POINTER TO AnyArrayUnbundleNode;
END_VAR
pAnyUnbundleNode := __NEW(AnyArrayUnbundleNode(ArrayDatatype := NodeDatatype));
CreateArrayUnbundleNode := pAnyUnbundleNode^;
END_METHOD

METHOD PROTECTED CreateDisplayNode : I_Node
VAR_INPUT
	NodeDatatype : I_Datatype;
END_VAR
VAR
	pAnyDisplayNode : POINTER TO AnyDisplayNode;
END_VAR
pAnyDisplayNode := __NEW(AnyDisplayNode(Datatype := NodeDatatype));
CreateDisplayNode := pAnyDisplayNode^;
END_METHOD

METHOD PROTECTED CreateLiteralNode : I_Node
VAR_INPUT
	NodeDatatype : I_Datatype;
END_VAR
VAR
	pAnyLiteralNode : POINTER TO AnyLiteralNode;
END_VAR
pAnyLiteralNode := __NEW(AnyLiteralNode(Datatype := NodeDatatype));
CreateLiteralNode := pAnyLiteralNode^;
END_METHOD

METHOD PROTECTED CreateStructureBundleNode : I_Node
VAR_INPUT
	NodeDatatype : I_StructuredDatatype;
END_VAR
VAR
	pAnyBundleNode : POINTER TO AnyStructureBundleNode;
END_VAR
pAnyBundleNode := __NEW(AnyStructureBundleNode(StructuredDatatype := NodeDatatype));
CreateStructureBundleNode := pAnyBundleNode^;
END_METHOD

METHOD PROTECTED CreateStructureUnbundleNode : I_Node
VAR_INPUT
	NodeDatatype : I_StructuredDatatype;
END_VAR
VAR
	pAnyUnbundleNode : POINTER TO AnyStructureUnbundleNode;
END_VAR
pAnyUnbundleNode := __NEW(AnyStructureUnbundleNode(StructuredDatatype := NodeDatatype));
CreateStructureUnbundleNode := pAnyUnbundleNode^;
END_METHOD

METHOD PRIVATE DeregisterWithDatatypes
VAR_INPUT
END_VAR
IF datatypes = 0 THEN
	RETURN;
END_IF

datatypes.OffEvent('OnDatatypeAdded',THIS^);
datatypes := 0;
END_METHOD

METHOD PRIVATE DisposeSelfCreatedNodes : BOOL
VAR
	node : I_Node;
END_VAR
WHILE selfCreatedNodes.TryPop(node) DO
	node.Dispose();
END_WHILE
END_METHOD

METHOD FB_exit : BOOL
VAR_INPUT
	bInCopyCode : BOOL; // if TRUE, the exit method is called for exiting an instance that is copied afterwards (online change).
END_VAR
IF bInCopyCode THEN
	RETURN;
END_IF

DeregisterWithDatatypes();
DisposeSelfCreatedNodes();
END_METHOD

METHOD FB_init : BOOL
VAR_INPUT
	bInitRetains : BOOL; // if TRUE, the retain variables are initialized (warm start / cold start)
	bInCopyCode : BOOL;  // if TRUE, the instance afterwards gets moved into the copy code (online change)
	Datatypes : I_Datatypes;
	NodeFactory : I_NodeFactory;	
END_VAR
THIS^.datatypes := Datatypes;
THIS^.nodeFactory := NodeFactory;

RegisterWithDatatypes();
END_METHOD

METHOD PUBLIC HandleEvent
VAR_INPUT
	Event : I_Event;
END_VAR
VAR
	datatypeAddedEvent : I_DatatypeAddedEvent;
	primativeDatatype : I_Datatype;
	aliasDatatypeAddedEvent : I_AliasDatatypeAddedEvent;
	aliasDatatype : I_AliasDatatype;
	enumDatatypeAddedEvent : I_EnumDatatypeAddedEvent;
	enumDatatype : I_EnumDatatype;
	structuredDatatypeAddedEvent : I_StructuredDatatypeAddedEvent;
	structureDatatype : I_StructuredDatatype;
	interfaceDatatypeAddedEvent : I_InterfaceDatatypeAddedEvent;
	interfaceDatatype : I_InterfaceDatatype;
	arrayDatatypeAddedEvent : I_ArrayDatatypeAddedEvent;
	arrayDatatype : I_ArrayDatatype;
END_VAR
IF __QUERYINTERFACE(event, aliasDatatypeAddedEvent) THEN
	aliasDatatype := aliasDatatypeAddedEvent.Target;
	RegisterUdtLiteralNodeOfType(aliasDatatype);
	RegisterUdtDisplayNodeOfType(aliasDatatype);
	
	// at this point we have the lowest level alias who's base type is not alias (or we reached a breakout)
	IF aliasDatatype.RootDatatype.TryResolveAsArrayDatatype(arrayDatatype) THEN
		RegisterAliasArrayBundleNodeOfType(aliasDatatype);
		RegisterAliasArrayUnbundleNodeOfType(aliasDatatype);
	ELSIF aliasDatatype.RootDatatype.TryResolveAsStructuredDatatype(structureDatatype) THEN
		RegisterAliasStructureBundleNodeOfType(aliasDatatype);
		RegisterAliasStructureUnbundleNodeOfType(aliasDatatype);
	END_IF
		
	RETURN;
END_IF

IF __QUERYINTERFACE(event, enumDatatypeAddedEvent) THEN
	enumDatatype := enumDatatypeAddedEvent.Target;
	RegisterUdtLiteralNodeOfType(enumDatatype);
	RegisterUdtDisplayNodeOfType(enumDatatype);
	RETURN;
END_IF

IF __QUERYINTERFACE(event, interfaceDatatypeAddedEvent) THEN
	interfaceDatatype := interfaceDatatypeAddedEvent.Target;
	RegisterInterfaceLiteralNodeOfType(interfaceDatatype);
	RegisterInterfaceDisplayNodeOfType(interfaceDatatype);
	RETURN;
END_IF

IF __QUERYINTERFACE(event, structuredDatatypeAddedEvent) THEN
	structureDatatype := structuredDatatypeAddedEvent.Target;
	RegisterUdtLiteralNodeOfType(structureDatatype);
	RegisterUdtDisplayNodeOfType(structureDatatype);
	RegisterStructureBundleNodeOfType(structureDatatype);
	RegisterStructureUnbundleNodeOfType(structureDatatype);
	RETURN;
END_IF

IF __QUERYINTERFACE(event, arrayDatatypeAddedEvent) THEN
	RegisterUdtLiteralNodeOfType(arrayDatatypeAddedEvent.Target);
	RegisterUdtDisplayNodeOfType(arrayDatatypeAddedEvent.Target);
	RegisterArrayBundleNodeOfType(arrayDatatypeAddedEvent.Target);
	RegisterArrayUnbundleNodeOfType(arrayDatatypeAddedEvent.Target);
	RETURN;
END_IF

IF __QUERYINTERFACE(event, datatypeAddedEvent) THEN
	primativeDatatype := datatypeAddedEvent.Target;
	RegisterPrimitiveLiteralNodeOfType(primativeDatatype);
	RegisterPrimitiveDisplayNodeOfType(primativeDatatype);
	RETURN;
END_IF
END_METHOD

METHOD PROTECTED RegisterAliasArrayBundleNodeOfType
VAR_INPUT
	AliasDatatype : I_AliasDatatype;
END_VAR
VAR
	node : I_Node;
	path : T_MAXSTRING;
END_VAR
node := CreateAliasArrayBundleNode(AliasDatatype);
selfCreatedNodes.Push(node);
path := concat('Bundle/', AliasDatatype.Identifier);
nodeFactory.AddNodeAsPrototype(path,node);
END_METHOD

METHOD PROTECTED RegisterAliasArrayUnbundleNodeOfType
VAR_INPUT
	AliasDatatype : I_AliasDatatype;
END_VAR
VAR
	node : I_Node;
	path : T_MAXSTRING;
END_VAR
node := CreateAliasArrayUnbundleNode(AliasDatatype);
selfCreatedNodes.Push(node);
path := concat('Unbundle/', AliasDatatype.Identifier);
nodeFactory.AddNodeAsPrototype(path,node);
END_METHOD

METHOD PROTECTED RegisterAliasStructureBundleNodeOfType
VAR_INPUT
	AliasDatatype : I_AliasDatatype;
END_VAR
VAR
	node : I_Node;
	path : T_MAXSTRING;
END_VAR
node := CreateAliasStructureBundleNode(AliasDatatype);
selfCreatedNodes.Push(node);
path := concat('Bundle/', AliasDatatype.Identifier);
nodeFactory.AddNodeAsPrototype(path,node);
END_METHOD

METHOD PROTECTED RegisterAliasStructureUnbundleNodeOfType
VAR_INPUT
	AliasDatatype : I_AliasDatatype;
END_VAR
VAR
	node : I_Node;
	path : T_MAXSTRING;
END_VAR
node := CreateAliasStructureUnbundleNode(AliasDatatype);
selfCreatedNodes.Push(node);
path := concat('Unbundle/', AliasDatatype.Identifier);
nodeFactory.AddNodeAsPrototype(path,node);
END_METHOD

METHOD PROTECTED RegisterArrayBundleNodeOfType
VAR_INPUT
	NodeDatatype : I_ArrayDatatype;
END_VAR
VAR
	node : I_Node;
	path : T_MAXSTRING;
END_VAR
node := CreateArrayBundleNode(NodeDatatype);
selfCreatedNodes.Push(node);
path := concat('Bundle/', NodeDatatype.Identifier);
nodeFactory.AddNodeAsPrototype(path,node);
END_METHOD

METHOD PROTECTED RegisterArrayUnbundleNodeOfType
VAR_INPUT
	NodeDatatype : I_ArrayDatatype;
END_VAR
VAR
	node : I_Node;
	path : T_MAXSTRING;
END_VAR
node := CreateArrayUnbundleNode(NodeDatatype);
selfCreatedNodes.Push(node);
path := concat('Unbundle/', NodeDatatype.Identifier);
nodeFactory.AddNodeAsPrototype(path,node);
END_METHOD

METHOD PROTECTED RegisterInterfaceDisplayNodeOfType
VAR_INPUT
	NodeDatatype : I_InterfaceDatatype;
END_VAR
VAR
	node : I_Node;
	path : T_MAXSTRING;
END_VAR
node := CreateDisplayNode(NodeDatatype);
selfCreatedNodes.Push(node);
path := concat('Display/', NodeDatatype.Identifier);
nodeFactory.AddNodeAsPrototype(path,node);
END_METHOD

METHOD PROTECTED RegisterInterfaceLiteralNodeOfType
VAR_INPUT
	NodeDatatype : I_InterfaceDatatype;
END_VAR
VAR
	node : I_Node;
	path : T_MAXSTRING;
END_VAR
node := CreateLiteralNode(NodeDatatype);
selfCreatedNodes.Push(node);
path := concat('Literal/', NodeDatatype.Identifier);
nodeFactory.AddNodeAsPrototype(path,node);
END_METHOD

METHOD PROTECTED RegisterPrimitiveDisplayNodeOfType
VAR_INPUT
	NodeDatatype : I_Datatype;
END_VAR
VAR
	node : I_Node;
	path : T_MAXSTRING;
END_VAR
node := CreateDisplayNode(NodeDatatype);
selfCreatedNodes.Push(node);
path := concat('Display/',NodeDatatype.TypeName);
nodeFactory.AddNodeAsPrototype(path,node);
END_METHOD

METHOD PROTECTED RegisterPrimitiveLiteralNodeOfType
VAR_INPUT
	NodeDatatype : I_Datatype;
END_VAR
VAR
	node : I_Node;
	path : T_MAXSTRING;
END_VAR
node := CreateLiteralNode(NodeDatatype);
selfCreatedNodes.Push(node);
path := concat('Literal/',NodeDatatype.TypeName);
nodeFactory.AddNodeAsPrototype(path,node);
END_METHOD

METHOD PROTECTED RegisterStructureBundleNodeOfType
VAR_INPUT
	NodeDatatype : I_StructuredDatatype;
END_VAR
VAR
	node : I_Node;
	path : T_MAXSTRING;
END_VAR
node := CreateStructureBundleNode(NodeDatatype);
selfCreatedNodes.Push(node);
path := concat('Bundle/', NodeDatatype.Identifier);
nodeFactory.AddNodeAsPrototype(path,node);
END_METHOD

METHOD PROTECTED RegisterStructureUnbundleNodeOfType
VAR_INPUT
	NodeDatatype : I_StructuredDatatype;
END_VAR
VAR
	node : I_Node;
	path : T_MAXSTRING;
END_VAR
node := CreateStructureUnbundleNode(NodeDatatype);
selfCreatedNodes.Push(node);
path := concat('Unbundle/', NodeDatatype.Identifier);
nodeFactory.AddNodeAsPrototype(path,node);
END_METHOD

METHOD PROTECTED RegisterUdtDisplayNodeOfType
VAR_INPUT
	NodeDatatype : I_UserDefinedDatatype;
END_VAR
VAR
	node : I_Node;
	path : T_MAXSTRING;
END_VAR
node := CreateDisplayNode(NodeDatatype);
selfCreatedNodes.Push(node);
path := concat('Display/', NodeDatatype.Identifier);
nodeFactory.AddNodeAsPrototype(path,node);
END_METHOD

METHOD PROTECTED RegisterUdtLiteralNodeOfType
VAR_INPUT
	NodeDatatype : I_UserDefinedDatatype;
END_VAR
VAR
	node : I_Node;
	path : T_MAXSTRING;
END_VAR
node := CreateLiteralNode(NodeDatatype);
selfCreatedNodes.Push(node);
path := concat('Literal/', NodeDatatype.Identifier);
nodeFactory.AddNodeAsPrototype(path,node);
END_METHOD

METHOD PRIVATE RegisterWithDatatypes
VAR_INPUT
END_VAR
IF datatypes = 0 THEN
	RETURN;
END_IF

datatypes.OnEvent('OnDatatypeAdded',THIS^);
END_METHOD

END_FUNCTION_BLOCK

// ---- Node/Bundle/AnyAliasArrayBundleNode.TcPOU
{attribute 'linkalways'} 
{attribute 'no_explicit_call' := 'This FB is a CLASS and must be accessed using methods or properties'}
{attribute 'enable_dynamic_creation'}
FUNCTION_BLOCK FINAL AnyAliasArrayBundleNode EXTENDS Node
VAR
	in : I_AliasDatatype;
	out : I_AliasDatatype;
	datatypeOperations : DatatypeOperations;
	selfMadeElements : Stack;
END_VAR

METHOD PUBLIC Clone : I_Node
VAR
	pNode : POINTER TO AnyAliasArrayBundleNode;
END_VAR
pNode := __NEW(AnyAliasArrayBundleNode(AliasDatatype := in));
Clone := pNode^;
END_METHOD

METHOD PRIVATE ConfigureFor1DArray
VAR_INPUT
	array1D : I_ArrayDatatype_1D;
END_VAR
VAR
	lowerBound : DINT;
	upperBound : DINT;
	i : DINT;
	element : I_Datatype;
	elementClone : I_Datatype;
END_VAR
IF NOT array1D.TryGetLowerBound(1, lowerBound) THEN
	RETURN;
END_IF

IF NOT array1D.TryGetUpperBound(1, upperBound) THEN
	RETURN;
END_IF

FOR i := lowerBound TO upperBound DO
	
	IF array1D.TryGetElementAsDatatypeByIndex(i, element) THEN
		elementClone := element.Clone();
		datatypeOperations.AddMemoryCopyOperation(elementClone, element);
		AddInput(Get1DIndexName(i), elementClone);
		selfMadeElements.Push(elementClone);
	END_IF
	
END_FOR
END_METHOD

METHOD PRIVATE ConfigureFor2DArray
VAR_INPUT
	array2D : I_ArrayDatatype_2D;
END_VAR
VAR
	lowerBoundD1 : DINT;
	upperBoundD1 : DINT;
	lowerBoundD2 : DINT;
	upperBoundD2 : DINT;
	i, j : DINT;
	element : I_Datatype;
	elementClone : I_Datatype;
END_VAR
IF NOT array2D.TryGetLowerBound(1, lowerBoundD1) THEN
	RETURN;
END_IF

IF NOT array2D.TryGetUpperBound(1, upperBoundD1) THEN
	RETURN;
END_IF

IF NOT array2D.TryGetLowerBound(2, lowerBoundD2) THEN
	RETURN;
END_IF

IF NOT array2D.TryGetUpperBound(2, upperBoundD2) THEN
	RETURN;
END_IF

FOR i := lowerBoundD1 TO upperBoundD1 DO
	FOR j := lowerBoundD2 TO upperBoundD2 DO
	
		IF array2D.TryGetElementAsDatatypeByIndex(i, j, element) THEN
			elementClone := element.Clone();
			datatypeOperations.AddMemoryCopyOperation(elementClone, element);
			AddInput(Get2DIndexName(i,j), elementClone);
			selfMadeElements.Push(elementClone);
		END_IF
	
	END_FOR
END_FOR
END_METHOD

METHOD PRIVATE ConfigureFor3DArray
VAR_INPUT
	array3D : I_ArrayDatatype_3D;
END_VAR
VAR
	lowerBoundD1 : DINT;
	upperBoundD1 : DINT;
	lowerBoundD2 : DINT;
	upperBoundD2 : DINT;
	lowerBoundD3 : DINT;
	upperBoundD3 : DINT;
	i, j, k : DINT;
	element : I_Datatype;
	elementClone : I_Datatype;
END_VAR
IF NOT array3D.TryGetLowerBound(1, lowerBoundD1) THEN
	RETURN;
END_IF

IF NOT array3D.TryGetUpperBound(1, upperBoundD1) THEN
	RETURN;
END_IF

IF NOT array3D.TryGetLowerBound(2, lowerBoundD2) THEN
	RETURN;
END_IF

IF NOT array3D.TryGetUpperBound(2, upperBoundD2) THEN
	RETURN;
END_IF

IF NOT array3D.TryGetLowerBound(3, lowerBoundD3) THEN
	RETURN;
END_IF

IF NOT array3D.TryGetUpperBound(3, upperBoundD3) THEN
	RETURN;
END_IF

FOR i := lowerBoundD1 TO upperBoundD1 DO
	FOR j := lowerBoundD2 TO upperBoundD2 DO
		FOR k := lowerBoundD3 TO upperBoundD3 DO
	
			IF array3D.TryGetElementAsDatatypeByIndex(i, j, k, element) THEN
				elementClone := element.Clone();
				datatypeOperations.AddMemoryCopyOperation(elementClone, element);
				AddInput(Get3DIndexName(i,j,k), elementClone);
				selfMadeElements.Push(elementClone);
			END_IF
			
		END_FOR
	END_FOR
END_FOR
END_METHOD

METHOD FB_exit : BOOL
VAR_INPUT
	bInCopyCode : BOOL; // if TRUE, the exit method is called for exiting an instance that is copied afterwards (online change).
END_VAR
VAR
	element : I_Datatype;
END_VAR
IF bInCopyCode THEN
	RETURN;
END_IF

in.Dispose();
out.Dispose();
datatypeOperations.Clear();

WHILE selfMadeElements.TryPop(element) DO
	IF element <> 0 THEN 
		element.dispose();
	END_IF
END_WHILE
END_METHOD

METHOD FB_init : BOOL
VAR_INPUT
	bInitRetains : BOOL; // if TRUE, the retain variables are initialized (warm start / cold start)
	bInCopyCode : BOOL;  // if TRUE, the instance afterwards gets moved into the copy code (online change)
	AliasDatatype : I_AliasDatatype;
END_VAR
VAR
	inAsArray : I_ArrayDatatype;
	inAs1D : I_ArrayDatatype_1D;
	inAs2D : I_ArrayDatatype_2D;
	inAs3D : I_ArrayDatatype_3D;
END_VAR
AliasDatatype.Clone().TryResolveAsAliasDatatype(out);
AddOutput('out', out);

AliasDatatype.Clone().TryResolveAsAliasDatatype(in);
in.RootDatatype.TryResolveAsArrayDatatype(inAsArray);

IF inAsArray.TryResolveAs1DArrayDatatype(inAs1D) THEN
	ConfigureFor1DArray(inAs1D);
ELSIF inAsArray.TryResolveAs2DArrayDatatype(inAs2D) THEN
	ConfigureFor2DArray(inAs2D);
ELSIF inAsArray.TryResolveAs3DArrayDatatype(inAs3D) THEN
	ConfigureFor3DArray(inAs3D);
END_IF
END_METHOD

METHOD PRIVATE Get1DIndexName : T_MAXSTRING
VAR_INPUT
	Index : DINT;
END_VAR
Get1DIndexName := concat('[',DINT_TO_STRING(Index));
Get1DIndexName := concat(Get1DIndexName,']');
END_METHOD

METHOD PRIVATE Get2DIndexName : T_MAXSTRING
VAR_INPUT
	Index1 : DINT;
	Index2 : DINT;
END_VAR
Get2DIndexName := concat('[',DINT_TO_STRING(Index1));
Get2DIndexName := concat(Get2DIndexName,',');
Get2DIndexName := concat(Get2DIndexName,DINT_TO_STRING(Index2));
Get2DIndexName := concat(Get2DIndexName,']');
END_METHOD

METHOD PRIVATE Get3DIndexName : T_MAXSTRING
VAR_INPUT
	Index1 : DINT;
	Index2 : DINT;
	Index3 : DINT;
END_VAR
Get3DIndexName := concat('[',DINT_TO_STRING(Index1));
Get3DIndexName := concat(Get3DIndexName,',');
Get3DIndexName := concat(Get3DIndexName,DINT_TO_STRING(Index2));
Get3DIndexName := concat(Get3DIndexName,',');
Get3DIndexName := concat(Get3DIndexName,DINT_TO_STRING(Index3));
Get3DIndexName := concat(Get3DIndexName,']');
END_METHOD

METHOD PROTECTED OnExecute : HRESULT
VAR
END_VAR
datatypeOperations.Execute();
memcpy(out.Address, in.Address, in.Size);
END_METHOD

END_FUNCTION_BLOCK

// ---- Node/Unbundle/AnyAliasArrayUnbundleNode.TcPOU
{attribute 'linkalways'} 
{attribute 'no_explicit_call' := 'This FB is a CLASS and must be accessed using methods or properties'}
{attribute 'enable_dynamic_creation'}
FUNCTION_BLOCK FINAL AnyAliasArrayUnbundleNode EXTENDS Node
VAR
	in : I_AliasDatatype;
	out : I_AliasDatatype;
	datatypeOperations : DatatypeOperations;
	selfMadeElements : Stack;
END_VAR

METHOD PUBLIC Clone : I_Node
VAR
	pNode : POINTER TO AnyAliasArrayUnbundleNode;
END_VAR
pNode := __NEW(AnyAliasArrayUnbundleNode(AliasDatatype := in));
Clone := pNode^;
END_METHOD

METHOD PRIVATE ConfigureFor1DArray
VAR_INPUT
	array1D : I_ArrayDatatype_1D;
END_VAR
VAR
	lowerBound : DINT;
	upperBound : DINT;
	i : DINT;
	element : I_Datatype;
	elementClone : I_Datatype;
END_VAR
IF NOT array1D.TryGetLowerBound(1, lowerBound) THEN
	RETURN;
END_IF

IF NOT array1D.TryGetUpperBound(1, upperBound) THEN
	RETURN;
END_IF

FOR i := lowerBound TO upperBound DO
	
	IF array1D.TryGetElementAsDatatypeByIndex(i, element) THEN
		elementClone := element.Clone();
		datatypeOperations.AddMemoryCopyOperation(element, elementClone);
		AddOutput(Get1DIndexName(i), elementClone);
		selfMadeElements.Push(elementClone);
	END_IF
	
END_FOR
END_METHOD

